// TwinCAT 3 PLC project LineaBosch5PLC
// Title: LineaBosch5
// Company: Normagrup
// ProjectVersion: 1.0
// ProgramVersion: 3.1.4023.0
// libraries:
//   Tc2_Standard, * (Beckhoff Automation GmbH)
//   Tc2_System, * (Beckhoff Automation GmbH)
//   Tc2_Utilities, * (Beckhoff Automation GmbH)
//   Tc3_Module, * (Beckhoff Automation GmbH)
// project tree:
//   DUTs/ ResultadoCiclo.TcDUT
//   GVLs/ GVL.TcGVL
//   / PlcTask.TcTTO
//   POUs/ ControlDescensoFin.TcPOU, ControlElevadorInicio.TcPOU, MAIN.TcPOU, PuestoAutomatico.TcPOU, PuestoTester.TcPOU, PuestoManual.TcPOU, PuestoManualV2.TcPOU, PuestoCupula.TcPOU, Seguridad.TcPOU
// real-time tasks:
//   TASK PlcTask: cycle T#10ms, priority 20, ADS port 350
//   TASK PlcTask1: cycle T#10ms, priority 21, ADS port 351
// I/O:
//   DEVICE Dispositivo 1 (EtherCAT), AmsNetId 5.97.60.79.2.1
//     CabeceraPLC [EK1200-5000 EtherCAT Power supply (2A E-Bus)]
//       Terminal 2 (EL1809) [EL1809 16Ch. Dig. Input 24V, 3ms]
//       Terminal 3 (EL2809) [EL2809 16Ch. Dig. Output 24V, 0.5A]
//       Terminal 4 (EK1110) [EK1110 EtherCAT extension]
//     FinlineaCinta [xFC01 - Rexroth mode]
//     FinLineaVertical [xFC01 - Rexroth mode]
//     CintaLineaSuperior [xFC01 - Rexroth mode]
//     Terminal89 [EK1100 EtherCAT Coupler (2A E-Bus)]
//       Terminal 9 (EL1809) [EL1809 16Ch. Dig. Input 24V, 3ms]
//       Terminal 10 (EL2809) [EL2809 16Ch. Dig. Output 24V, 0.5A]
//       Terminal 31 (EL9011) [EL9011 End Terminal]
//     Valvulas89 [EX260-SEC3 EtherCAT SI Unit (16DO_PNP) Rev1.2]
//     Terminal67 [EK1100 EtherCAT Coupler (2A E-Bus)]
//       Terminal 13 (EL1809) [EL1809 16Ch. Dig. Input 24V, 3ms]
//       Terminal 14 (EL2809) [EL2809 16Ch. Dig. Output 24V, 0.5A]
//       Terminal 32 (EL9011) [EL9011 End Terminal]
//     Valvulas67 [EX260-SEC3 EtherCAT SI Unit (16DO_PNP) Rev1.2]
//     Terminal45 [EK1100 EtherCAT Coupler (2A E-Bus)]
//       Terminal 17 (EL1809) [EL1809 16Ch. Dig. Input 24V, 3ms]
//       Terminal 18 (EL2809) [EL2809 16Ch. Dig. Output 24V, 0.5A]
//       Terminal 33 (EL9011) [EL9011 End Terminal]
//     Valvulas45 [EX260-SEC3 EtherCAT SI Unit (16DO_PNP) Rev1.2]
//     Terminales23 [EK1100 EtherCAT Coupler (2A E-Bus)]
//       Terminal 21 (EL1809) [EL1809 16Ch. Dig. Input 24V, 3ms]
//       Terminal 22 (EL2809) [EL2809 16Ch. Dig. Output 24V, 0.5A]
//       Terminal 34 (EL9011) [EL9011 End Terminal]
//     Valvulas23 [EX260-SEC3 EtherCAT SI Unit (16DO_PNP) Rev1.2]
//     Terminal1 [EK1100 EtherCAT Coupler (2A E-Bus)]
//       Terminal 25 (EL2809) [EL2809 16Ch. Dig. Output 24V, 0.5A]
//       Terminal 26 (EL1809) [EL1809 16Ch. Dig. Input 24V, 3ms]
//       Terminal 35 (EL9011) [EL9011 End Terminal]
//     InicioLineaCinta [xFC01 - Rexroth mode]
//     InicioLineaVertical [xFC01 - Rexroth mode]
//     CintaLineaInferior [xFC01 - Rexroth mode]
//     Valvulas1 [EX260-SEC3 EtherCAT SI Unit (16DO_PNP) Rev1.2]
//   DEVICE Dispositivo 4 (NOV-DP-RAM)
//   DEVICE Dispositivo 6 (RT-Ethernet Protocol), AmsNetId 5.97.60.79.7.1
// variable links:
//   LineaBosch5PLC/LineaBosch5PLC Instance <-> Device 1 (EtherCAT)/CabeceraPLC/Term 2 (EL1809)
//     PlcTask Inputs/GVL.ElevadorFinLinea.PresenciaCintaAbajo <-> Channel 6/Input
//     PlcTask Inputs/GVL.ElevadorFinLinea.PresenciaCintaArriba <-> Channel 7/Input
//     PlcTask Inputs/GVL.ElevadorFinLinea.PulsadorBajar <-> Channel 4/Input
//     PlcTask Inputs/GVL.ElevadorFinLinea.PulsadorSubir <-> Channel 3/Input
//     PlcTask Inputs/GVL.ElevadorFinLinea.SensorAbajo <-> Channel 9/Input
//     PlcTask Inputs/GVL.ElevadorFinLinea.SensorArriba <-> Channel 8/Input
//     PlcTask Inputs/GVL.Elevadorfin1_Presencia <-> Channel 12/Input
//     PlcTask Inputs/GVL.Elevadorfin2_Presencia <-> Channel 14/Input
//     PlcTask Inputs/MAIN.ControlSeguridad.CuadroPrincipalAutomatico <-> Channel 1/Input
//     PlcTask Inputs/MAIN.ControlSeguridad.CuadroPrincipalRunStop <-> Channel 2/Input
//     PlcTask Inputs/MAIN.ControlSeguridad.SeguridadSetas <-> Channel 5/Input
//   LineaBosch5PLC/LineaBosch5PLC Instance <-> Device 1 (EtherCAT)/CabeceraPLC/Term 3 (EL2809)
//     PlcTask Outputs/GVL.SemaforoAmarillo <-> Channel 14/Output
//     PlcTask Outputs/GVL.SemaforoRojo <-> Channel 15/Output
//     PlcTask Outputs/GVL.SemaforoVerde <-> Channel 16/Output
//   LineaBosch5PLC/LineaBosch5PLC Instance <-> Device 1 (EtherCAT)/CintaLineaInferior
//     PlcTask Outputs/MAIN.ControlSeguridad.MotorInferior_Command <-> RxPDO5/Control Word
//     PlcTask Outputs/MAIN.ControlSeguridad.MotorInferior_Freq <-> RxPDO5/Frequency Command
//   LineaBosch5PLC/LineaBosch5PLC Instance <-> Device 1 (EtherCAT)/CintaLineaSuperior
//     PlcTask Outputs/MAIN.ControlSeguridad.MotorSuperior_Command <-> RxPDO5/Control Word
//     PlcTask Outputs/MAIN.ControlSeguridad.MotorSuperior_Freq <-> RxPDO5/Frequency Command
//   LineaBosch5PLC/LineaBosch5PLC Instance <-> Device 1 (EtherCAT)/FinLineaVertical
//     PlcTask Outputs/GVL.ElevadorFinLinea.MotorElevacion_Command <-> RxPDO5/Control Word
//     PlcTask Outputs/GVL.ElevadorFinLinea.MotorElevacion_Freq <-> RxPDO5/Frequency Command
//   LineaBosch5PLC/LineaBosch5PLC Instance <-> Device 1 (EtherCAT)/FinlineaCinta
//     PlcTask Outputs/GVL.ElevadorFinLinea.MotorExtraccion_Command <-> RxPDO5/Control Word
//     PlcTask Outputs/GVL.ElevadorFinLinea.MotorExtraccion_Freq <-> RxPDO5/Frequency Command
//   LineaBosch5PLC/LineaBosch5PLC Instance <-> Device 1 (EtherCAT)/InicioLineaCinta
//     PlcTask Outputs/GVL.ElevadorInicioLinea.MotorExtraccion_Command <-> RxPDO5/Control Word
//     PlcTask Outputs/GVL.ElevadorInicioLinea.MotorExtraccion_Freq <-> RxPDO5/Frequency Command
//   LineaBosch5PLC/LineaBosch5PLC Instance <-> Device 1 (EtherCAT)/InicioLineaVertical
//     PlcTask Outputs/GVL.ElevadorInicioLinea.MotorElevacion_Command <-> RxPDO5/Control Word
//     PlcTask Outputs/GVL.ElevadorInicioLinea.MotorElevacion_Freq <-> RxPDO5/Frequency Command
//   LineaBosch5PLC/LineaBosch5PLC Instance <-> Device 1 (EtherCAT)/Terminal1/Term 26 (EL1809)
//     PlcTask Inputs/GVL.ElevadorInicioLinea.PresenciaCintaAbajo <-> Channel 10/Input
//     PlcTask Inputs/GVL.ElevadorInicioLinea.PresenciaCintaArriba <-> Channel 9/Input
//     PlcTask Inputs/GVL.ElevadorInicioLinea.PulsadorBajar <-> Channel 2/Input
//     PlcTask Inputs/GVL.ElevadorInicioLinea.PulsadorSubir <-> Channel 1/Input
//     PlcTask Inputs/GVL.ElevadorInicioLinea.SensorAbajo <-> Channel 4/Input
//     PlcTask Inputs/GVL.ElevadorInicioLinea.SensorArriba <-> Channel 3/Input
//     PlcTask Inputs/GVL.ElevadorInicioLinea.SensorPaletEnEspera <-> Channel 7/Input
//     PlcTask Inputs/GVL.Elevadorinicio1_Presencia <-> Channel 6/Input
//     PlcTask Inputs/GVL.Elevadorinicio2_Presencia <-> Channel 8/Input
//     PlcTask Inputs/GVL.Puesto11_Presencia <-> Channel 11/Input
//     PlcTask Inputs/GVL.Puesto12_Presencia <-> Channel 13/Input
//   LineaBosch5PLC/LineaBosch5PLC Instance <-> Device 1 (EtherCAT)/Terminal45/Term 17 (EL1809)
//     PlcTask Inputs/GVL.Puesto41_Presencia <-> Channel 3/Input
//     PlcTask Inputs/GVL.Puesto42_Presencia <-> Channel 4/Input
//     PlcTask Inputs/GVL.Puesto51_Presencia <-> Channel 11/Input
//     PlcTask Inputs/GVL.Puesto52_Presencia <-> Channel 12/Input
//   LineaBosch5PLC/LineaBosch5PLC Instance <-> Device 1 (EtherCAT)/Terminal67/Term 13 (EL1809)
//     PlcTask Inputs/GVL.Puesto61_Presencia <-> Channel 3/Input
//     PlcTask Inputs/GVL.Puesto62_Presencia <-> Channel 4/Input
//     PlcTask Inputs/GVL.Puesto71_Presencia <-> Channel 11/Input
//     PlcTask Inputs/GVL.Puesto72_Presencia <-> Channel 12/Input
//     PlcTask Inputs/GVL.Puesto71_Bypass <-> Channel 9/Input
//     PlcTask Inputs/GVL.Puesto71_Pulsador <-> Channel 10/Input
//     PlcTask Inputs/GVL.Puesto72.Fail <-> Channel 13/Input
//     PlcTask Inputs/GVL.Puesto72.Pass <-> Channel 14/Input
//     PlcTask Inputs/GVL.Puesto72.SelectorByPass <-> Channel 15/Input
//     PlcTask Inputs/GVL.Puesto72_PresenciaPieza <-> Channel 16/Input
//   LineaBosch5PLC/LineaBosch5PLC Instance <-> Device 1 (EtherCAT)/Terminal67/Term 14 (EL2809)
//     PlcTask Outputs/GVL.Puesto72.Ready <-> Channel 9/Output
//     PlcTask Outputs/GVL.Puesto72_Actuador <-> Channel 10/Output
//   LineaBosch5PLC/LineaBosch5PLC Instance <-> Device 1 (EtherCAT)/Terminal89/Term 10 (EL2809)
//     PlcTask Outputs/GVL.Puesto81.LuzRoja <-> Channel 1/Output
//   LineaBosch5PLC/LineaBosch5PLC Instance <-> Device 1 (EtherCAT)/Terminal89/Term 9 (EL1809)
//     PlcTask Inputs/GVL.Puesto81_Presencia <-> Channel 3/Input
//     PlcTask Inputs/GVL.Puesto82_Presencia <-> Channel 4/Input
//     PlcTask Inputs/GVL.Puesto91_Presencia <-> Channel 12/Input
//     PlcTask Inputs/GVL.Puesto92_Presencia <-> Channel 11/Input
//     PlcTask Inputs/GVL.Puesto81_Pulsador <-> Channel 5/Input
//   LineaBosch5PLC/LineaBosch5PLC Instance <-> Device 1 (EtherCAT)/Terminales23/Term 21 (EL1809)
//     PlcTask Inputs/GVL.Puesto21_Presencia <-> Channel 3/Input
//     PlcTask Inputs/GVL.Puesto22_Presencia <-> Channel 4/Input
//     PlcTask Inputs/GVL.Puesto31_Presencia <-> Channel 11/Input
//     PlcTask Inputs/GVL.Puesto32_Presencia <-> Channel 12/Input
//   LineaBosch5PLC/LineaBosch5PLC Instance <-> Device 1 (EtherCAT)/Valvulas1
//     PlcTask Outputs/GVL.TerminalValvulas1 <-> Byte 0/Output
//   LineaBosch5PLC/LineaBosch5PLC Instance <-> Device 1 (EtherCAT)/Valvulas23
//     PlcTask Outputs/GVL.TerminalValvulas23 <-> Byte 0/Output
//   LineaBosch5PLC/LineaBosch5PLC Instance <-> Device 1 (EtherCAT)/Valvulas45
//     PlcTask Outputs/GVL.TerminalValvulas45 <-> Byte 0/Output
//   LineaBosch5PLC/LineaBosch5PLC Instance <-> Device 1 (EtherCAT)/Valvulas67
//     PlcTask Outputs/GVL.TerminalValvulas67 <-> Byte 0/Output
//     PlcTask Outputs/GVL.TerminalValvulas67_2 <-> Byte 1/Output
//   LineaBosch5PLC/LineaBosch5PLC Instance <-> Device 1 (EtherCAT)/Valvulas89
//     PlcTask Outputs/GVL.TerminalValvulas89 <-> Byte 0/Output

CONFIGURATION LineaBosch5PLC
    RESOURCE PLC ON TwinCAT3
        TASK PlcTask(INTERVAL := T#10ms, PRIORITY := 21);
        PROGRAM MAIN WITH PlcTask : MAIN;
    END_RESOURCE
END_CONFIGURATION

// ---- DUTs/ResultadoCiclo.TcDUT
{attribute 'pack_mode' := '1'}
TYPE ResultadoCiclo :
STRUCT
	producto  : STRING[25];
	ciclo: INT;
	hora: DT;
	FalloPuesto: ARRAY[1..18] OF BOOL;
	RetrasoPuesto: ARRAY[1..18] OF INT;
END_STRUCT
END_TYPE

// ---- GVLs/GVL.TcGVL
VAR_GLOBAL
	
	
	SeguridadOK :BOOL;
	ModoRun: BOOL;
	ModoAutomatico :BOOL;
	ModoDobleCarga :BOOL := FALSE;
	
	SemaforoRojo AT %Q* :BOOL;
	SemaforoAmarillo AT %Q* :BOOL;
	SemaforoVerde AT %Q* :BOOL;
	
	FinTiempo :BOOL;
	FinCiclo:BOOL;
	
	TiempoDeCiclo: INT := 20;   //segundos de tiempo de ciclo
	VelocidadCinta: UINT := 50; //Velocidad motores cinta en hercios

	FalloPallet: ARRAY[1..18] OF BOOL;

	HoraActual :DT;
	fbLocalTime     : FB_LocalSystemTime;

	
	
	
	TerminalValvulas1 AT %Q*: USINT;
	TerminalValvulas23 AT %Q* : USINT;
	TerminalValvulas45 AT %Q*: USINT;
	TerminalValvulas67 AT %Q* : USINT;
	TerminalValvulas67_2 AT %Q* : USINT;
	TerminalValvulas89 AT %Q* : USINT;
			
	
	Puesto11_Centrador AT %Q* :BOOL;
	Puesto11_stoper AT %Q*:BOOL;
	Puesto12_centrador AT %Q*: BOOL; 
	Puesto12_stoper AT %Q*:BOOL;
	Puesto21_centrador AT %Q*: BOOL; 
	Puesto21_stoper AT %Q*:BOOL;
	Puesto22_centrador AT %Q*: BOOL; 
	Puesto22_stoper AT %Q*:BOOL;
	Puesto31_centrador AT %Q*: BOOL; 
	Puesto31_stoper AT %Q*:BOOL;
	Puesto32_centrador AT %Q*: BOOL; 
	Puesto32_stoper AT %Q*:BOOL;
	Puesto41_centrador AT %Q*: BOOL; 
	Puesto41_stoper AT %Q*:BOOL;
	Puesto42_centrador AT %Q*: BOOL; 
	Puesto42_stoper AT %Q*:BOOL;
	Puesto51_centrador AT %Q*: BOOL; 
	Puesto51_stoper AT %Q*:BOOL;
	Puesto52_centrador AT %Q*: BOOL; 
	Puesto52_stoper AT %Q*:BOOL;
	Puesto61_centrador AT %Q*: BOOL; 
	Puesto61_stoper AT %Q*:BOOL;
	Puesto62_centrador AT %Q*: BOOL; 
	Puesto62_stoper AT %Q*:BOOL;
	Puesto71_centrador AT %Q*: BOOL; 
	Puesto71_stoper AT %Q*:BOOL;
	Puesto72_centrador AT %Q*: BOOL; 
	Puesto72_stoper AT %Q*:BOOL;
	Puesto81_centrador AT %Q*: BOOL; 
	Puesto81_stoper AT %Q*:BOOL;
	Puesto82_centrador AT %Q*: BOOL; 
	Puesto82_stoper AT %Q*:BOOL;
	Puesto91_centrador AT %Q*: BOOL; 
	Puesto91_stoper AT %Q*:BOOL;
	Puesto92_centrador AT %Q*: BOOL; 
	Puesto92_stoper AT %Q*:BOOL;
	
	Puesto71_Actuador AT %Q* :BOOL;
	Puesto72_Actuador AT %Q* :BOOL;
	Puesto72_LuzVerde AT %Q* :BOOL;
	

	
	Puesto11_Presencia AT %I* :BOOL;
	Puesto12_Presencia AT %I* :BOOL;
	Puesto21_Presencia AT %I* :BOOL;
	Puesto22_Presencia AT %I* :BOOL;
	Puesto31_Presencia AT %I* :BOOL;
	Puesto32_Presencia AT %I* :BOOL;
	Puesto41_Presencia AT %I* :BOOL;
	Puesto42_Presencia AT %I* :BOOL;
	Puesto51_Presencia AT %I* :BOOL;
	Puesto52_Presencia AT %I* :BOOL;
	Puesto61_Presencia AT %I* :BOOL;
	Puesto62_Presencia AT %I* :BOOL;
	Puesto71_Presencia AT %I* :BOOL;
	Puesto72_Presencia AT %I* :BOOL;
	Puesto81_Presencia AT %I* :BOOL;
	Puesto82_Presencia AT %I* :BOOL;
	Puesto91_Presencia AT %I* :BOOL;
	Puesto92_Presencia AT %I* :BOOL;
	
	Puesto61_Bypass AT %I* :BOOL;
	Puesto71_Pulsador AT %I* :BOOL;
	Puesto71_Bypass AT %I* :BOOL;
	Puesto72_PresenciaPieza AT %I* :BOOL;
	Puesto81_Pulsador AT %I* :BOOL;

	Elevadorinicio1_Presencia AT %I* :BOOL;
	Elevadorinicio2_Presencia AT %I* :BOOL;
	Elevadorfin1_Presencia AT %I* :BOOL;
	Elevadorfin2_Presencia AT %I* :BOOL;

	
	Puesto11: PuestoManual;
    Puesto12: PuestoManual;
    Puesto21: PuestoManual;
    Puesto22: PuestoManual;
    Puesto31: PuestoManual;
	Puesto32: PuestoManual;
    Puesto41: PuestoManual;
	Puesto42: PuestoManual;
    Puesto51: PuestoManual;
	Puesto52: PuestoManual;
    Puesto61: PuestoManual;
	Puesto62: PuestoManual;
    Puesto71: PuestoCupula;
	Puesto72: PuestoAutomatico;
    Puesto81: PuestoManual;
	Puesto82: PuestoManual;
    Puesto91: PuestoManual;
	Puesto92: PuestoManualV2;
	

	

	ElevadorFinLinea: ControlDescensoFin;
	ElevadorInicioLinea: ControlElevadorInicio;
	
END_VAR

VAR_GLOBAL PERSISTENT
	Producto : STRING[30] := 'SINDEFINIR';
	Est_Resultados : ARRAY[1..3000] OF ResultadoCiclo;
	PunteroEst: INT := 1;
END_VAR

// ---- POUs/MAIN.TcPOU
PROGRAM MAIN
VAR
	ControlSeguridad: Seguridad;
	ElevadorFinLleno : BOOL;
	ElevadorInicioLleno :BOOL;
	ElevadorInicioPuedeExtraer :BOOL;
	FalloTest :BOOL;

	fbTime   : FB_LocalSystemTime := ( bEnable := TRUE, dwCycle := 100 );
	
	Semaforo: USINT;
	EstadoPuestos: DINT;
	
END_VAR

	
ControlSeguridad();
fbTime();
gvl.HoraActual := SYSTEMTIME_TO_DT(fbTime.systemTime);

///PUESTO 1 -----------------------------------

Puesto12 ( Enable:= gvl.ModoRun, Reset := FALSE,SensorPallet:= gvl.Puesto12_Presencia, 
		Centrador => gvl.Puesto12_centrador, StopperOFF => gvl.Puesto12_stoper,
FinCiclo := gvl.FinCiclo, NumeroDePuesto :=1   );


///PUESTO 2 -----------------------------------
Puesto21 ( Enable:= gvl.ModoRun, Reset := FALSE,SensorPallet:= gvl.Puesto21_Presencia, 
		Centrador => gvl.Puesto21_centrador, StopperOFF => gvl.Puesto21_stoper,
FinCiclo := gvl.FinCiclo, NumeroDePuesto :=2   );
Puesto22 ( Enable:= gvl.ModoRun, Reset := FALSE,SensorPallet:= gvl.Puesto22_Presencia, 
		Centrador => gvl.Puesto22_centrador, StopperOFF => gvl.Puesto22_stoper,
FinCiclo := gvl.FinCiclo, NumeroDePuesto :=3   );

///PUESTO 3 -----------------------------------
Puesto31 ( Enable:= gvl.ModoRun, Reset := FALSE,SensorPallet:= gvl.Puesto31_Presencia, 
		Centrador => gvl.Puesto31_centrador, StopperOFF => gvl.Puesto31_stoper,
FinCiclo := gvl.FinCiclo, NumeroDePuesto :=4   );
Puesto32 ( Enable:= gvl.ModoRun, Reset := FALSE,SensorPallet:= gvl.Puesto32_Presencia, 
		Centrador => gvl.Puesto32_centrador, StopperOFF => gvl.Puesto32_stoper,
FinCiclo := gvl.FinCiclo, NumeroDePuesto :=5   );

///PUESTO 4 -----------------------------------
Puesto41 ( Enable:= gvl.ModoRun, Reset := FALSE,SensorPallet:= gvl.Puesto41_Presencia, 
		Centrador => gvl.Puesto41_centrador, StopperOFF => gvl.Puesto41_stoper,
FinCiclo := gvl.FinCiclo, NumeroDePuesto :=6   );
Puesto42 ( Enable:= gvl.ModoRun, Reset := FALSE,SensorPallet:= gvl.Puesto42_Presencia, 
		Centrador => gvl.Puesto42_centrador, StopperOFF => gvl.Puesto42_stoper,
FinCiclo := gvl.FinCiclo, NumeroDePuesto :=7   );

///PUESTO 5 -----------------------------------
Puesto51 ( Enable:= gvl.ModoRun, Reset := FALSE,SensorPallet:= gvl.Puesto51_Presencia, 
		Centrador => gvl.Puesto51_centrador, StopperOFF => gvl.Puesto51_stoper,
FinCiclo := gvl.FinCiclo, NumeroDePuesto :=8   );
Puesto52 ( Enable:= gvl.ModoRun, Reset := FALSE,SensorPallet:= gvl.Puesto52_Presencia, 
		Centrador => gvl.Puesto52_centrador, StopperOFF => gvl.Puesto52_stoper,
FinCiclo := gvl.FinCiclo, NumeroDePuesto :=9   );

///PUESTO 6 -----------------------------------
Puesto61 ( Enable:= gvl.ModoRun, Reset := FALSE,SensorPallet:= gvl.Puesto61_Presencia, 
		Centrador => gvl.Puesto61_centrador, StopperOFF => gvl.Puesto61_stoper,
FinCiclo := gvl.FinCiclo, NumeroDePuesto :=10   );
Puesto62 ( Enable:= gvl.ModoRun, Reset := FALSE,SensorPallet:= gvl.Puesto62_Presencia, 
		Centrador => gvl.Puesto62_centrador, StopperOFF => gvl.Puesto62_stoper,
FinCiclo := gvl.FinCiclo, NumeroDePuesto :=11   );

///PUESTO 7 -----------------------------------
//Puesto71 ( Enable:= gvl.ModoRun, Reset := FALSE,SensorPallet:= gvl.Puesto71_Presencia, 
//		Centrador => gvl.Puesto71_centrador, StopperOFF => gvl.Puesto71_stoper,
//FinCiclo := gvl.FinCiclo, NumeroDePuesto :=12   );

///*****************************************************

Puesto71 ( Enable:= gvl.ModoRun, Reset :=FALSE,SensorPallet:= gvl.Puesto71_Presencia, 
			sensorpieza1 :=TRUE, SelectorByPass := gvl.Puesto71_Bypass,
		Centrador => gvl.Puesto71_centrador, StopperOFF => gvl.Puesto71_stoper,
		FinCiclo := gvl.FinCiclo , NumeroDePuesto :=12  );
gvl.Puesto71_Actuador:= Puesto71.Actuador;

//***********************************************************



//Puesto del Test 
Puesto72 ( Enable:= gvl.ModoRun, Reset :=FALSE,SensorPallet:= gvl.Puesto72_Presencia, 
			sensorpieza1 := gvl.Puesto72_presenciapieza, Centrador => gvl.Puesto72_centrador, StopperOFF => gvl.Puesto72_stoper,
		FinCiclo := gvl.FinCiclo , NumeroDePuesto :=13  );
gvl.Puesto72_Actuador := gvl.Puesto72.Ready; ///gvl.Puesto72_centrador AND gvl.Puesto72_PresenciaPieza ;
gvl.Puesto72_LuzVerde := Puesto72.Ready;


///PUESTO 8 -----------------------------------
Puesto81 ( Enable:= gvl.ModoRun, Reset := FALSE,SensorPallet:= gvl.Puesto81_Presencia, 
		Centrador => gvl.Puesto81_centrador, StopperOFF => gvl.Puesto81_stoper,
		pulsador1:= gvl.Puesto81_Pulsador,
FinCiclo := gvl.FinCiclo, NumeroDePuesto :=14   );

Puesto82 ( Enable:= gvl.ModoRun, Reset := FALSE,SensorPallet:= gvl.Puesto82_Presencia, 
		Centrador => gvl.Puesto82_centrador, StopperOFF => gvl.Puesto82_stoper,
FinCiclo := gvl.FinCiclo, NumeroDePuesto :=15  );


///PUESTO 9 -----------------------------------
Puesto91 ( Enable:= gvl.ModoRun, Reset := FALSE,SensorPallet:= gvl.Puesto91_Presencia, 
		Centrador => gvl.Puesto91_centrador, StopperOFF => gvl.Puesto91_stoper,
FinCiclo := gvl.FinCiclo, NumeroDePuesto :=16   );



/// ojo modo doble carga 
gvl.ModoDobleCarga := TRUE;

Puesto11 ( Enable:= gvl.ModoRun, Reset := FALSE,SensorPallet:= gvl.Puesto11_Presencia, 
		Centrador => gvl.Puesto11_centrador, StopperOFF => gvl.Puesto11_stoper,
FinCiclo := gvl.FinCiclo, NumeroDePuesto :=17  );


Puesto92 ( Enable:= gvl.ModoRun, Reset := FALSE,SensorPallet:= gvl.Puesto92_Presencia, 
		Centrador => gvl.Puesto92_centrador, StopperOFF => gvl.Puesto92_stoper,
FinCiclo := gvl.FinCiclo, NumeroDePuesto :=18 , ModoDoble := gvl.ModoDobleCarga  );


/// CONTROL ELEVADORES

IF gvl.ModoDobleCarga = TRUE THEN
	ElevadorFinLleno := gvl.Elevadorfin1_Presencia AND gvl.Elevadorfin2_Presencia;
	ElevadorInicioLleno := gvl.Elevadorinicio1_Presencia AND gvl.Elevadorinicio2_Presencia;
	ElevadorInicioPuedeExtraer := Puesto11.EsperandoPalet AND Puesto12.EsperandoPalet;
ELSE
	ElevadorFinLleno := gvl.Elevadorfin1_Presencia;
	ElevadorInicioLleno := gvl.Elevadorinicio1_Presencia;
	ElevadorInicioPuedeExtraer := Puesto11.EsperandoPalet;
END_IF

ElevadorInicioLinea( Enabled:= gvl.ModoRun, SeguridadOK:= GVL.SeguridadOK,
					SensorPaletFuera := Puesto11.SensorPallet,
					SensorPaletDentro := ElevadorInicioLleno,
					 PuedeExtraer := Puesto11.EsperandoPalet AND NOT Puesto12.EsperandoPalet);
					 
ElevadorFinLinea( Enabled:= gvl.ModoRun, SeguridadOK:= GVL.SeguridadOK, 
				SensorPaletDentro := ElevadorFinLleno,
				SensorPaletFuera := gvl.Elevadorfin2_Presencia,
				PuedeExtraer := TRUE);

TerminalValvulas1.0 := ElevadorInicioLinea.StopperOFF;
TerminalValvulas1.1 := gvl.Puesto11_stoper;
TerminalValvulas1.2 := gvl.Puesto12_stoper;
TerminalValvulas1.3 := gvl.Puesto11_centrador;
TerminalValvulas1.4 := gvl.Puesto12_centrador;

TerminalValvulas23.0 := gvl.Puesto21_stoper;
TerminalValvulas23.1 := gvl.Puesto22_stoper;
TerminalValvulas23.2 := gvl.Puesto31_stoper;
TerminalValvulas23.3 := gvl.Puesto32_stoper;
TerminalValvulas23.4 := gvl.Puesto21_centrador;
TerminalValvulas23.5 := gvl.Puesto22_centrador;
TerminalValvulas23.6 := gvl.Puesto31_centrador;
TerminalValvulas23.7 := gvl.Puesto32_centrador;

TerminalValvulas45.0 := gvl.Puesto41_stoper;
TerminalValvulas45.1 := gvl.Puesto42_stoper;
TerminalValvulas45.2 := gvl.Puesto51_stoper;
TerminalValvulas45.3 := gvl.Puesto52_stoper;
TerminalValvulas45.4 := gvl.Puesto41_centrador;
TerminalValvulas45.5 := gvl.Puesto42_centrador;
TerminalValvulas45.6 := gvl.Puesto51_centrador;
TerminalValvulas45.7 := gvl.Puesto52_centrador;

TerminalValvulas67.0 := gvl.Puesto61_stoper;
TerminalValvulas67.1 := gvl.Puesto62_stoper;
TerminalValvulas67.2 := gvl.Puesto71_stoper;
TerminalValvulas67.3 := gvl.Puesto72_stoper;
TerminalValvulas67.4 := gvl.Puesto61_centrador;
TerminalValvulas67.5 := gvl.Puesto62_centrador;
TerminalValvulas67.6 := gvl.Puesto71_centrador;
TerminalValvulas67.7 := gvl.Puesto72_centrador;
TerminalValvulas67_2.0 := gvl.Puesto72_actuador;
TerminalValvulas67_2.1 := gvl.Puesto71_actuador;


TerminalValvulas89.0 := gvl.Puesto81_stoper;
TerminalValvulas89.1 := gvl.Puesto82_stoper;
TerminalValvulas89.2 := gvl.Puesto91_stoper;
TerminalValvulas89.3 := gvl.Puesto92_stoper;
TerminalValvulas89.4 := gvl.Puesto81_centrador;
TerminalValvulas89.5 := gvl.Puesto82_centrador;
TerminalValvulas89.6 := gvl.Puesto91_centrador;
TerminalValvulas89.7 := gvl.Puesto92_centrador;

/// Variables para el HMI
Semaforo.0 := gvl.SemaforoRojo;
Semaforo.1 := gvl.SemaforoAmarillo;
Semaforo.2 := gvl.SemaforoVerde;

 EstadoPuestos.0 := GVL.ElevadorInicioLinea.Ready;
 EstadoPuestos.1 := GVL.Puesto11.FinPuesto;
 EstadoPuestos.2 := GVL.Puesto12.FinPuesto;
 EstadoPuestos.3 := GVL.Puesto21.FinPuesto;
 EstadoPuestos.4 := GVL.Puesto22.FinPuesto ;
 EstadoPuestos.5 := GVL.Puesto31.FinPuesto;
 EstadoPuestos.6 := GVL.Puesto32.FinPuesto;
 EstadoPuestos.7 := GVL.Puesto41.FinPuesto;
 EstadoPuestos.8 := GVL.Puesto42.FinPuesto ;
 EstadoPuestos.9 := GVL.Puesto51.FinPuesto ;
 EstadoPuestos.10 := GVL.Puesto52.FinPuesto ;
 EstadoPuestos.11 := GVL.Puesto61.FinPuesto ;
 EstadoPuestos.12 := GVL.Puesto62.FinPuesto ;
 EstadoPuestos.13 := GVL.Puesto71.FinPuesto ;
 EstadoPuestos.14 := GVL.Puesto72.FinPuesto ;
 EstadoPuestos.15 := GVL.Puesto81.FinPuesto ;
 EstadoPuestos.16 := GVL.Puesto82.FinPuesto ;
 EstadoPuestos.17 := GVL.Puesto91.FinPuesto ;
 EstadoPuestos.18 := GVL.Puesto92.FinPuesto ;
 EstadoPuestos.19 := GVL.ElevadorFinLinea.Ready;

END_PROGRAM

// ---- POUs/Seguridad.TcPOU
FUNCTION_BLOCK Seguridad
VAR_INPUT
	
	CuadroPrincipalRunStop AT%I*:BOOL;
	CuadroPrincipalAutomatico AT%I*:BOOL;
	SeguridadSetas AT%I*:BOOL;
END_VAR
VAR_OUTPUT
	CuadroLedVerde AT%Q*:BOOL;
	CuadroLedAmarillo AT%Q*:BOOL;
	
	MotorSuperior_Freq  AT%Q*: UINT;
	MotorSuperior_Command AT%Q*: INT;
		
	MotorInferior_Freq  AT%Q*: UINT;
	MotorInferior_Command AT%Q*: INT;
	
	LineaReady :BOOL;
	FinTiempoTON :TON;
	
	
	
END_VAR
VAR
	FlancoRunStop:R_TRIG;
	TempCiclo:TON;
	TempRetraso:TON;
	Resultados : ResultadoCiclo;

	puesto: INT;
	Falso: BOOL;
END_VAR

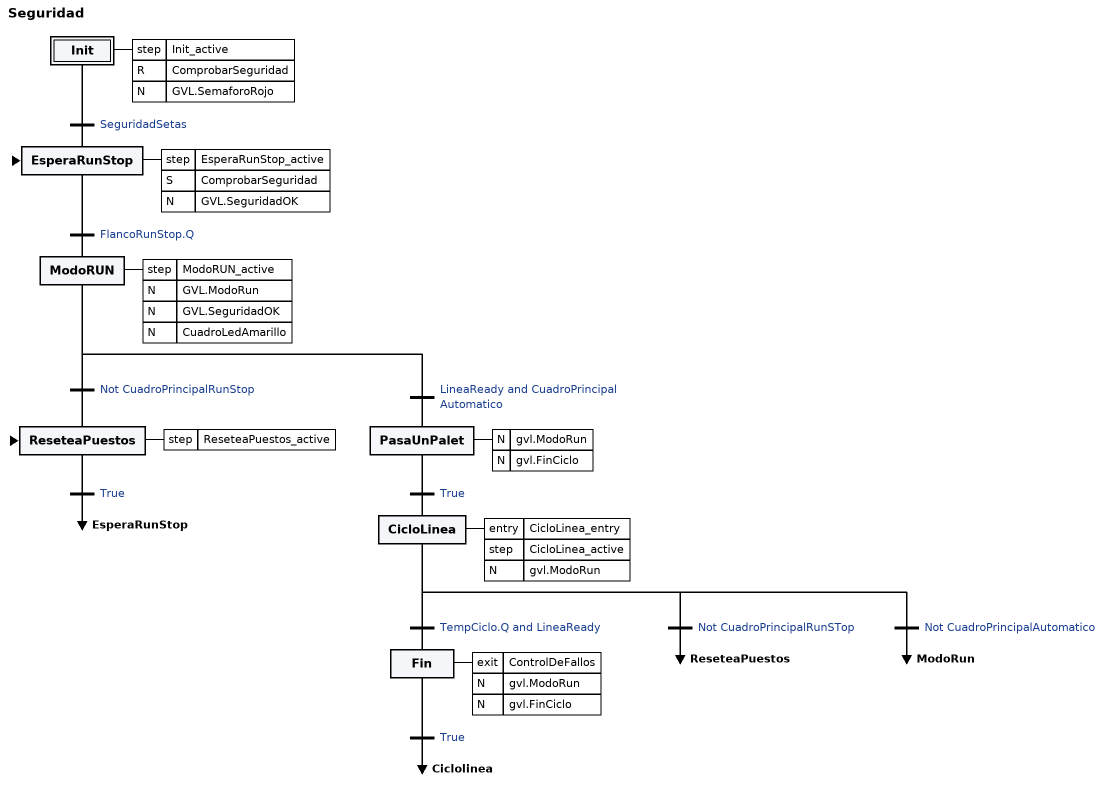
INITIAL_STEP Init:
    Init_active(N);  // step action
    ComprobarSeguridad(R);
    GVL.SemaforoRojo(N);
END_STEP
TRANSITION FROM Init TO EsperaRunStop
    := SeguridadSetas;
END_TRANSITION
STEP EsperaRunStop:  // min time T#1s
    EsperaRunStop_active(N);  // step action
    ComprobarSeguridad(S);
    GVL.SeguridadOK(N);
END_STEP
TRANSITION FROM EsperaRunStop TO ModoRUN
    := FlancoRunStop.Q;
END_TRANSITION
STEP ModoRUN:  // min time T#1s
    ModoRUN_active(N);  // step action
    GVL.ModoRun(N);
    GVL.SeguridadOK(N);
    CuadroLedAmarillo(N);
END_STEP
TRANSITION FROM ModoRUN TO ReseteaPuestos
    := Not CuadroPrincipalRunStop;
END_TRANSITION
STEP ReseteaPuestos:  // min time T#1s
    ReseteaPuestos_active(N);  // step action
END_STEP
TRANSITION FROM ReseteaPuestos TO EsperaRunStop
    := True;
END_TRANSITION
TRANSITION FROM ModoRUN TO PasaUnPalet
    := LineaReady and CuadroPrincipalAutomatico;
END_TRANSITION
STEP PasaUnPalet:  // min time T#3s
    gvl.ModoRun(N);
    gvl.FinCiclo(N);
END_STEP
TRANSITION FROM PasaUnPalet TO CicloLinea
    := True;
END_TRANSITION
STEP CicloLinea:  // min time T#4s
    CicloLinea_entry(P1);  // entry action
    CicloLinea_active(N);  // step action
    gvl.ModoRun(N);
END_STEP
TRANSITION FROM CicloLinea TO Fin
    := TempCiclo.Q and LineaReady;
END_TRANSITION
STEP Fin:  // min time T#3s
    ControlDeFallos(P0);  // exit action
    gvl.ModoRun(N);
    gvl.FinCiclo(N);
END_STEP
TRANSITION FROM Fin TO Ciclolinea
    := True;
END_TRANSITION
TRANSITION FROM CicloLinea TO ReseteaPuestos
    := Not CuadroPrincipalRunSTop;
END_TRANSITION
TRANSITION FROM CicloLinea TO ModoRun
    := Not CuadroPrincipalAutomatico;
END_TRANSITION

ACTION CicloLinea_active:
TempCiclo(IN:=TRUE);
TempRetraso(IN:=TempCiclo.Q);

gvl.SemaforoVerde := TRUE;

IF (    (ElevadorInicioLinea.Ready OR gvl.ModoDobleCarga)///no esperamos por elevador inicio en modo doble carga
	AND (ElevadorFinLinea.ready OR GVL.Puesto92.EsperandoPalet ) //si el ultimo  puesto no tieen palet no esperamos por elevador fin
	AND GVL.Puesto11.FinPuesto AND
		GVL.Puesto12.FinPuesto AND
		GVL.Puesto21.FinPuesto AND
		GVL.Puesto22.FinPuesto AND
		GVL.Puesto31.FinPuesto AND
		GVL.Puesto32.FinPuesto AND
		GVL.Puesto41.FinPuesto AND
		GVL.Puesto42.FinPuesto AND
		GVL.Puesto51.FinPuesto AND
		GVL.Puesto52.FinPuesto AND
		GVL.Puesto61.FinPuesto AND
		GVL.Puesto62.FinPuesto AND
		GVL.Puesto71.FinPuesto AND
		GVL.Puesto72.FinPuesto AND
		GVL.Puesto81.FinPuesto AND
		GVL.Puesto82.FinPuesto AND
		GVL.Puesto91.FinPuesto AND
		(gvl.Puesto81.LuzRoja = FALSE) AND
		(GVL.Puesto92.FinPuesto OR gvl.ModoDobleCarga))
THEN
		LineaReady := TRUE;
		gvl.SemaforoAmarillo :=  FALSE;
ELSE 
	    LineaReady := FALSE;
		gvl.SemaforoAmarillo := TempCiclo.Q;
END_IF


IF TempCiclo.Q AND NOT Lineaready THEN

		IF NOT  GVL.Puesto11.FinPuesto THEN gvl.Est_Resultados[gvl.PunteroEst].RetrasoPuesto[1] := TIME_TO_INT(TempRetraso.ET)/1000; END_IF 
		IF NOT 	GVL.Puesto12.FinPuesto THEN gvl.Est_Resultados[gvl.PunteroEst].RetrasoPuesto[2] := TIME_TO_INT(TempRetraso.ET); END_IF 
		if not 	GVL.Puesto21.FinPuesto then gvl.Est_Resultados[gvl.PunteroEst].RetrasoPuesto[3] := TIME_TO_INT(TempRetraso.ET); END_IF 
		if not 	GVL.Puesto22.FinPuesto then gvl.Est_Resultados[gvl.PunteroEst].RetrasoPuesto[4] := TIME_TO_INT(TempRetraso.ET); END_IF 
		if not 	GVL.Puesto31.FinPuesto then gvl.Est_Resultados[gvl.PunteroEst].RetrasoPuesto[5] := TIME_TO_INT(TempRetraso.ET); END_IF 
		if not 	GVL.Puesto32.FinPuesto then gvl.Est_Resultados[gvl.PunteroEst].RetrasoPuesto[6] := TIME_TO_INT(TempRetraso.ET); END_IF 
		if not 	GVL.Puesto41.FinPuesto then gvl.Est_Resultados[gvl.PunteroEst].RetrasoPuesto[7] := TIME_TO_INT(TempRetraso.ET); END_IF 
		if not 	GVL.Puesto42.FinPuesto then gvl.Est_Resultados[gvl.PunteroEst].RetrasoPuesto[8] := TIME_TO_INT(TempRetraso.ET); END_IF 
		if not 	GVL.Puesto51.FinPuesto then gvl.Est_Resultados[gvl.PunteroEst].RetrasoPuesto[9] := TIME_TO_INT(TempRetraso.ET); END_IF 
		if not 	GVL.Puesto52.FinPuesto then gvl.Est_Resultados[gvl.PunteroEst].RetrasoPuesto[10] := TIME_TO_INT(TempRetraso.ET); END_IF 
		if not 	GVL.Puesto61.FinPuesto then gvl.Est_Resultados[gvl.PunteroEst].RetrasoPuesto[11] := TIME_TO_INT(TempRetraso.ET); END_IF 
		if not 	GVL.Puesto62.FinPuesto then gvl.Est_Resultados[gvl.PunteroEst].RetrasoPuesto[12] := TIME_TO_INT(TempRetraso.ET); END_IF 
		if not 	GVL.Puesto71.FinPuesto then gvl.Est_Resultados[gvl.PunteroEst].RetrasoPuesto[13] := TIME_TO_INT(TempRetraso.ET); END_IF 
		if not 	GVL.Puesto72.FinPuesto then gvl.Est_Resultados[gvl.PunteroEst].RetrasoPuesto[14] := TIME_TO_INT(TempRetraso.ET); END_IF 
		if not 	GVL.Puesto81.FinPuesto then gvl.Est_Resultados[gvl.PunteroEst].RetrasoPuesto[15] := TIME_TO_INT(TempRetraso.ET); END_IF 
		if not 	GVL.Puesto82.FinPuesto then gvl.Est_Resultados[gvl.PunteroEst].RetrasoPuesto[16] := TIME_TO_INT(TempRetraso.ET); END_IF 
		if not 	GVL.Puesto91.FinPuesto then gvl.Est_Resultados[gvl.PunteroEst].RetrasoPuesto[17] := TIME_TO_INT(TempRetraso.ET); END_IF 
		if not 	GVL.Puesto92.FinPuesto then gvl.Est_Resultados[gvl.PunteroEst].RetrasoPuesto[18] := TIME_TO_INT(TempRetraso.ET); END_IF 

END_IF
END_ACTION

ACTION CicloLinea_entry:
TempCiclo(IN:=FALSE, PT:= DWORD_TO_TIME(  (INT_TO_DWORD(gvl.TiempoDeCiclo) -3)* 1000));
TempRetraso(IN:=FALSE, PT:= T#15M);



gvl.PunteroEst := gvl.PunteroEst +1;
IF gvl.PunteroEst > 1999 THEN
	gvl.PunteroEst := 1;
END_IF


//Creamos un nuevo registros
gvl.Est_Resultados[gvl.PunteroEst].Ciclo := gvl.TiempoDeCiclo;
gvl.Est_Resultados[gvl.PunteroEst].Producto := gvl.Producto;
gvl.Est_Resultados[gvl.PunteroEst].hora := gvl.HoraActual;



FOR puesto := 1 TO 18 DO
	gvl.Est_Resultados[gvl.PunteroEst].FalloPuesto[puesto] := FALSE;
	gvl.Est_Resultados[gvl.PunteroEst].RetrasoPuesto[puesto] := 0;
	
END_FOR
END_ACTION

ACTION ComprobarSeguridad:
IF NOT SeguridadSetas THEN
	SFCReset:=TRUE;
END_IF
END_ACTION

ACTION ControlDeFallos:




//avanzamos el fallo en el palet y guardamos estadistica
FOR puesto := 18 TO 2 BY -1 DO
	gvl.Est_Resultados[gvl.PunteroEst].FalloPuesto[puesto] := gvl.FalloPallet[puesto];
	gvl.FalloPallet[puesto] := gvl.FalloPallet[puesto -1 ];
END_FOR

gvl.FalloPallet[1] := Falso;
END_ACTION

ACTION EsperaRunStop_active:
FlancoRunStop(CLK:=CuadroPrincipalRunStop);

Gvl.SemaforoAmarillo := TRUE;
MotorCintaSuperior(0);
MotorCintaInferior(0);
END_ACTION

ACTION Init_active:
MotorCintaSuperior(0);
MotorCintaInferior(0);
SFCreset := FALSE;
gvl.SemaforoAmarillo :=FALSE;
gvl.SemaforoVerde := FALSE;
END_ACTION

ACTION ModoRUN_active:

TempCiclo(IN:=FALSE);

IF ElevadorFinLinea.Ready THEN
 MotorCintaSuperior(1);
END_IF

gvl.SemaforoAmarillo :=TRUE;

IF ElevadorInicioLinea.EsperandoPalet OR ElevadorInicioLinea.Ready THEN
	MotorCintaInferior(1);
END_IF

IF (ElevadorInicioLinea.Ready AND
	ElevadorFinLinea.ready AND 
	GVL.Puesto12.FinPuesto AND
	GVL.Puesto21.FinPuesto AND
	GVL.Puesto22.FinPuesto AND
	GVL.Puesto31.FinPuesto AND
	GVL.Puesto32.FinPuesto AND
	GVL.Puesto41.FinPuesto AND
	GVL.Puesto42.FinPuesto AND
	GVL.Puesto51.FinPuesto AND
	GVL.Puesto52.FinPuesto AND
	GVL.Puesto61.FinPuesto AND
	GVL.Puesto62.FinPuesto AND
	GVL.Puesto71.FinPuesto AND
	GVL.Puesto72.FinPuesto AND
	GVL.Puesto81.FinPuesto AND
	GVL.Puesto82.FinPuesto AND
	GVL.Puesto91.FinPuesto )
THEN		
		gvl.SemaforoVerde := TRUE;
		LineaReady := TRUE;
			
ELSE
			LineaReady:=FALSE;
			gvl.FinTiempo :=FALSE;
			gvl.SemaforoVerde := FALSE;
END_IF
END_ACTION

METHOD PRIVATE MotorCintaInferior : BOOL
VAR_INPUT
	Direccion: INT;
END_VAR
MotorInferior_Freq := gvl.VelocidadCinta * 100;


MotorInferior_Command := 0;
MotorInferior_Command.7 := 1 ; //Control Word Active


IF Direccion  = 0 THEN
	MotorInferior_Command.3 := 1 ; // Stop according to parameter setting	

ELSIF gvl.ElevadorInicioLinea.PresenciaCintaAbajo AND NOT gvl.ElevadorInicioLinea.SensorAbajo THEN
	// presencia en la salida y el elevador no esta abajo: paramos y ERROR
	MotorInferior_Command.3 := 1 ;
	
ELSIF Direccion  = 1 THEN		
		MotorInferior_Command.2 := 1 ; //1 reversed 0 fordward
		MotorInferior_Command.0 := 1 ; // Run Command active
ELSE
	MotorInferior_Command.3 := 1 ; // Stop according to parameter setting	
END_IF
END_METHOD

METHOD PRIVATE MotorCintaSuperior : BOOL
VAR_INPUT
	Direccion: INT;
END_VAR
MotorSuperior_Freq := gvl.VelocidadCinta * 100;


MotorSuperior_Command := 0;
MotorSuperior_Command.7 := 1 ; //Control Word Active

IF Direccion = 0 THEN
	MotorSuperior_Command.3 := 1 ; // Stop according to parameter setting	
ELSIF gvl.Elevadorfinlinea.PresenciaCintaArriba AND NOT gvl.Elevadorfinlinea.sensorarriba THEN
	//ERROR : palet en la salida y elevador no arriba
	MotorSuperior_Command.3 := 1 ;
ELSIF Direccion  = 1 THEN		
		MotorSuperior_Command.2 := 0 ; //1 reversed 0 fordward
		MotorSuperior_Command.0 := 1 ; // Run Command active
ELSE
	MotorSuperior_Command.3 := 1 ; // Stop according to parameter setting	
END_IF
END_METHOD

ACTION ReseteaPuestos_active:

//Resetea los puestos para pasar un palet


GVL.Puesto11.SFCreset := TRUE;
GVL.Puesto12.SFCreset := TRUE;
GVL.Puesto21.SFCreset := TRUE;
GVL.Puesto22.SFCreset := TRUE;
GVL.Puesto31.sfcreset := TRUE;
GVL.Puesto32.sfcreset := TRUE;
GVL.Puesto41.sfcreset := TRUE;
GVL.Puesto42.sfcreset := TRUE;
GVL.Puesto51.sfcreset := TRUE;
GVL.Puesto52.sfcreset := TRUE;
GVL.Puesto61.sfcreset := TRUE;
GVL.Puesto62.sfcreset := TRUE;
GVL.Puesto71.sfcreset := TRUE;
GVL.Puesto72.sfcreset := TRUE;
GVL.Puesto81.sfcreset := TRUE;
GVL.Puesto82.sfcreset := TRUE;
GVL.Puesto91.sfcreset := TRUE;
GVL.Puesto92.sfcreset := TRUE;

ElevadorInicioLinea.SFCreset := TRUE;
ElevadorFinLinea.SFCreset := TRUE;
END_ACTION

END_FUNCTION_BLOCK

// ---- POUs/PuestoManual.TcPOU
FUNCTION_BLOCK PuestoManual
VAR_INPUT
	SFCreset:BOOL;
	Reset:BOOL;
	Enable:BOOL;
	FinCiclo:BOOL;
	SensorPallet:BOOL;
	Pulsador1 AT %I*:BOOL;
	NumeroDePuesto :INT;
	
END_VAR
VAR_OUTPUT
	StopperOFF AT %Q*:BOOL;
	Centrador AT%Q*:BOOL;
	LuzRoja AT%Q*:BOOL;
	FinPuesto:BOOL;
	SalidaAlarma:BOOL;
	EnMovimiento:BOOL;
	EsperandoPalet :BOOL;
	RetrasoPuesto :INT;
END_VAR
VAR
END_VAR

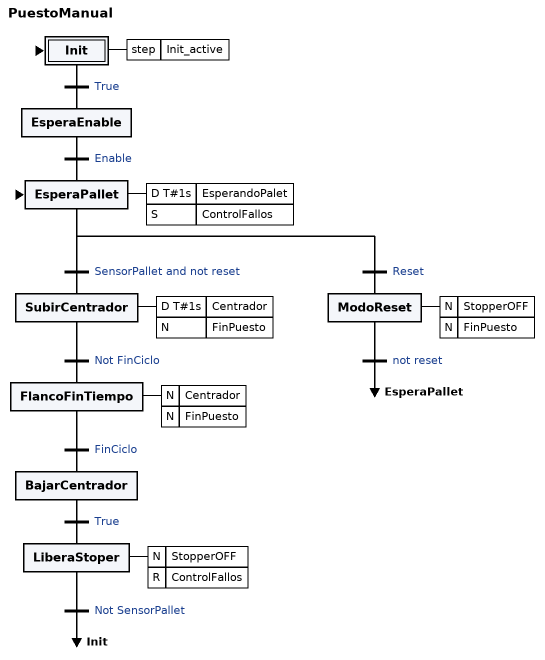
INITIAL_STEP Init:
    Init_active(N);  // step action
END_STEP
TRANSITION FROM Init TO EsperaEnable
    := True;
END_TRANSITION
STEP EsperaEnable:
END_STEP
TRANSITION FROM EsperaEnable TO EsperaPallet
    := Enable;
END_TRANSITION
STEP EsperaPallet:
    EsperandoPalet(D, T#1s);
    ControlFallos(S);
END_STEP
TRANSITION FROM EsperaPallet TO SubirCentrador
    := SensorPallet and not reset;
END_TRANSITION
STEP SubirCentrador:  // min time T#1s
    Centrador(D, T#1s);
    FinPuesto(N);
END_STEP
TRANSITION FROM SubirCentrador TO FlancoFinTiempo
    := Not FinCiclo;
END_TRANSITION
STEP FlancoFinTiempo:
    Centrador(N);
    FinPuesto(N);
END_STEP
TRANSITION FROM FlancoFinTiempo TO BajarCentrador
    := FinCiclo;
END_TRANSITION
STEP BajarCentrador:  // min time T#1s
END_STEP
TRANSITION FROM BajarCentrador TO LiberaStoper
    := True;
END_TRANSITION
TRANSITION FROM EsperaPallet TO ModoReset
    := Reset;
END_TRANSITION
STEP ModoReset:
    StopperOFF(N);
    FinPuesto(N);
END_STEP
TRANSITION FROM ModoReset TO EsperaPallet
    := not reset;
END_TRANSITION
STEP LiberaStoper:  // min time T#1s
    StopperOFF(N);
    ControlFallos(R);
END_STEP
TRANSITION FROM LiberaStoper TO Init
    := Not SensorPallet;
END_TRANSITION

ACTION ControlFallos:

IF GVL.FalloPallet[NumeroDePuesto] THEN
	LuzRoja :=TRUE;
	FinPuesto := FALSE;
ELSE
	LuzRoja :=FALSE;
	FinPuesto := TRUE;
END_IF


IF GVL.FalloPallet[NumeroDePuesto] AND Pulsador1 THEN
	GVL.FalloPallet[NumeroDePuesto] := FALSE;
END_IF
END_ACTION

ACTION Init_active:
LuzRoja := FALSE;
FinPUesto :=FALSE;
SFCreset:=FALSE;
END_ACTION

END_FUNCTION_BLOCK

// ---- POUs/PuestoCupula.TcPOU
FUNCTION_BLOCK PuestoCupula
VAR_INPUT
	Reset:BOOL;
	SFCreset:BOOL;
	Enable:BOOL;
	FinCiclo:BOOL;
	SensorPallet:BOOL;
	Pulsador1 AT %I*:BOOL;
	NumeroDePuesto :INT;	
	SelectorByPass AT %I*:BOOL;
	Pass AT %I*:BOOL;
	Fail AT %I*:BOOL;
	
	SensorPieza1 AT %I*:BOOL;
	SensorPieza2 AT %I*:BOOL;
	
	SensorCupulaAtras AT%I*:BOOL;

END_VAR
VAR_OUTPUT
	
	Ready AT %Q*:BOOL;
	StopperOFF AT %Q*:BOOL;
	Centrador AT%Q*:BOOL;
	Actuador AT%Q*:BOOL;
	LuzAmbar AT%Q*:BOOL;
	SalidaAlarma:BOOL;
	EnMovimiento:BOOL;
	EsperandoPalet:BOOL;
	RetrasoPuesto :INT;
	FinPuesto:BOOL;
	
	CupulaAdelante AT%Q*:BOOL;
	CupulaAtras AT%Q*:BOOL;

	
	
END_VAR

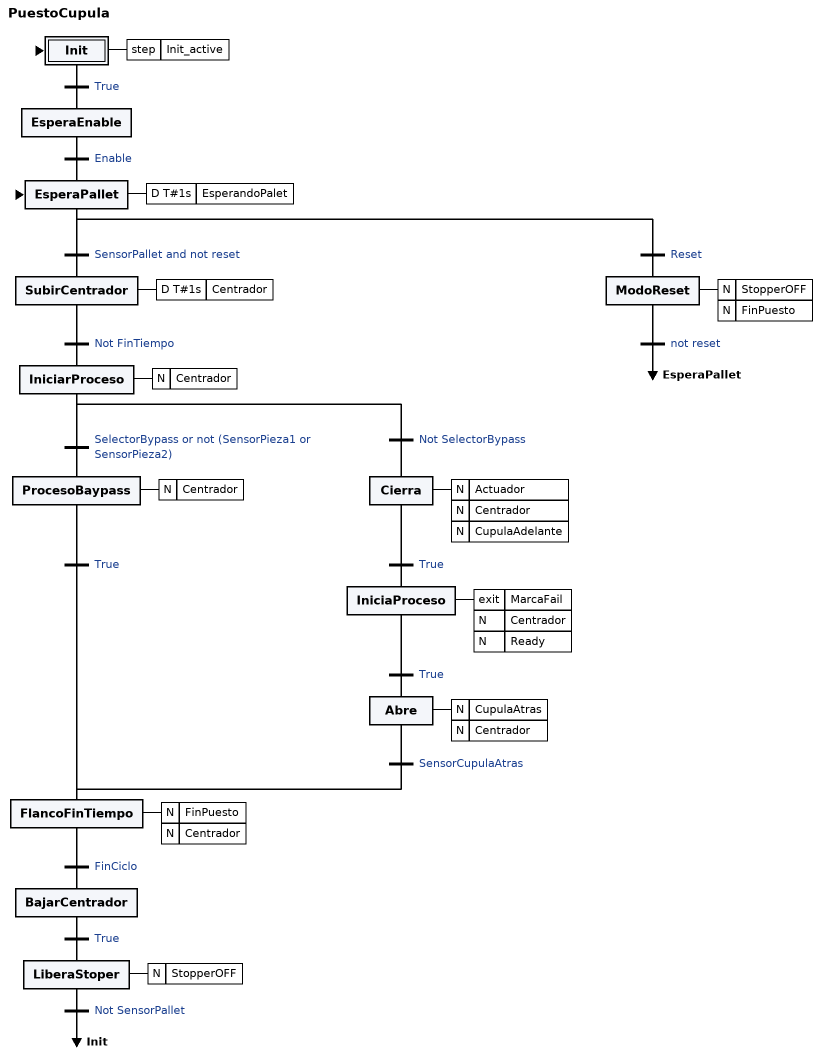
INITIAL_STEP Init:
    Init_active(N);  // step action
END_STEP
TRANSITION FROM Init TO EsperaEnable
    := True;
END_TRANSITION
STEP EsperaEnable:
END_STEP
TRANSITION FROM EsperaEnable TO EsperaPallet
    := Enable;
END_TRANSITION
STEP EsperaPallet:
    EsperandoPalet(D, T#1s);
END_STEP
TRANSITION FROM EsperaPallet TO SubirCentrador
    := SensorPallet and not reset;
END_TRANSITION
STEP SubirCentrador:  // min time T#2s
    Centrador(D, T#1s);
END_STEP
TRANSITION FROM SubirCentrador TO IniciarProceso
    := Not FinTiempo;
END_TRANSITION
STEP IniciarProceso:
    Centrador(N);
END_STEP
TRANSITION FROM IniciarProceso TO ProcesoBaypass
    := SelectorBypass or not (SensorPieza1 or SensorPieza2);
END_TRANSITION
STEP ProcesoBaypass:
    Centrador(N);
END_STEP
TRANSITION FROM ProcesoBaypass TO FlancoFinTiempo
    := True;
END_TRANSITION
TRANSITION FROM IniciarProceso TO Cierra
    := Not SelectorBypass;
END_TRANSITION
STEP Cierra:  // min time T#5s
    Actuador(N);
    Centrador(N);
    CupulaAdelante(N);
END_STEP
TRANSITION FROM Cierra TO IniciaProceso
    := True;
END_TRANSITION
STEP IniciaProceso:  // min time T#5s
    MarcaFail(P0);  // exit action
    Centrador(N);
    Ready(N);
END_STEP
TRANSITION FROM IniciaProceso TO Abre
    := True;
END_TRANSITION
STEP Abre:
    CupulaAtras(N);
    Centrador(N);
END_STEP
TRANSITION FROM Abre TO FlancoFinTiempo
    := SensorCupulaAtras;
END_TRANSITION
STEP FlancoFinTiempo:
    FinPuesto(N);
    Centrador(N);
END_STEP
TRANSITION FROM FlancoFinTiempo TO BajarCentrador
    := FinCiclo;
END_TRANSITION
STEP BajarCentrador:  // min time T#1s
END_STEP
TRANSITION FROM BajarCentrador TO LiberaStoper
    := True;
END_TRANSITION
TRANSITION FROM EsperaPallet TO ModoReset
    := Reset;
END_TRANSITION
STEP ModoReset:
    StopperOFF(N);
    FinPuesto(N);
END_STEP
TRANSITION FROM ModoReset TO EsperaPallet
    := not reset;
END_TRANSITION
STEP LiberaStoper:  // min time T#1s
    StopperOFF(N);
END_STEP
TRANSITION FROM LiberaStoper TO Init
    := Not SensorPallet;
END_TRANSITION

ACTION EsperaEnable_active:

END_ACTION

ACTION Init_active:
FinPUesto :=FALSE;
SFCreset:=FALSE;
END_ACTION

ACTION MarcaFail:
IF  Fail = TRUE THEN 
	gvl.FalloPallet[NumeroDePuesto] := TRUE;
END_IF
END_ACTION

END_FUNCTION_BLOCK

// ---- POUs/PuestoAutomatico.TcPOU
FUNCTION_BLOCK PuestoAutomatico
VAR_INPUT
	Reset:BOOL;
	SFCreset:BOOL;
	Enable:BOOL;
	FinCiclo:BOOL;
	SensorPallet:BOOL;
	Pulsador1 AT %I*:BOOL;

	NumeroDePuesto :INT;
	
	SelectorByPass AT %I*:BOOL;
	Pass AT %I*:BOOL;
	Fail AT %I*:BOOL;
	
	SensorPieza1 AT %I*:BOOL;
	SensorPieza2 AT %I*:BOOL;
	
END_VAR
VAR_OUTPUT
	
	Ready AT %Q*:BOOL;
	StopperOFF AT %Q*:BOOL;
	Centrador AT%Q*:BOOL;
	LuzAmbar AT%Q*:BOOL;
	SalidaAlarma:BOOL;
	EnMovimiento:BOOL;
	EsperandoPalet:BOOL;
	RetrasoPuesto :INT;
	FinPuesto:BOOL;
	
	
	
END_VAR
VAR
END_VAR

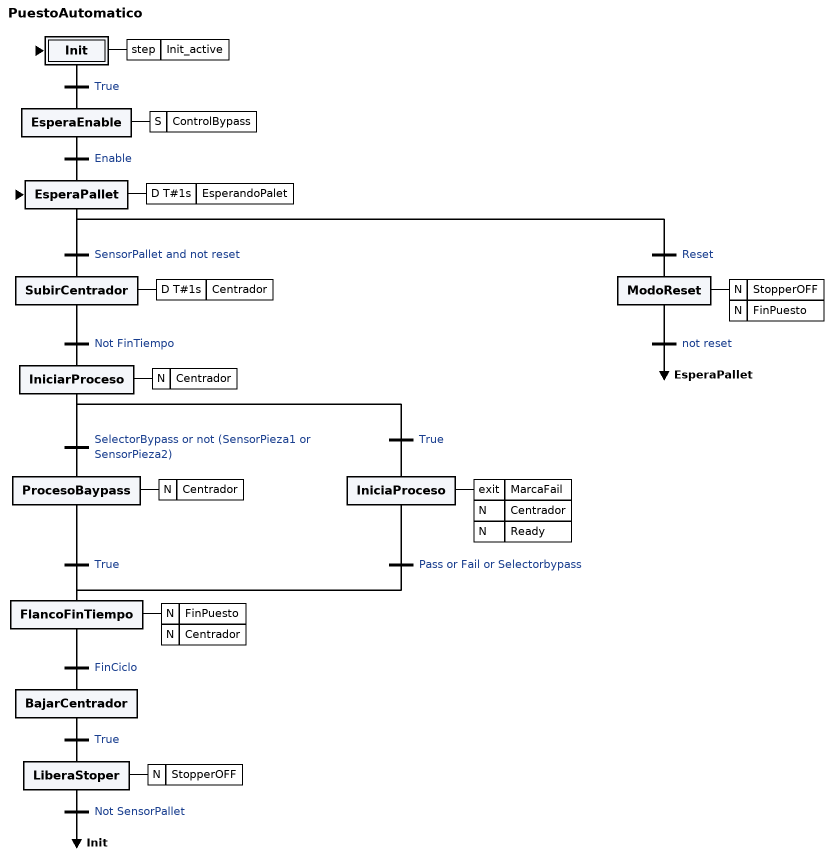
INITIAL_STEP Init:
    Init_active(N);  // step action
END_STEP
TRANSITION FROM Init TO EsperaEnable
    := True;
END_TRANSITION
STEP EsperaEnable:
    ControlBypass(S);
END_STEP
TRANSITION FROM EsperaEnable TO EsperaPallet
    := Enable;
END_TRANSITION
STEP EsperaPallet:
    EsperandoPalet(D, T#1s);
END_STEP
TRANSITION FROM EsperaPallet TO SubirCentrador
    := SensorPallet and not reset;
END_TRANSITION
STEP SubirCentrador:  // min time T#2s
    Centrador(D, T#1s);
END_STEP
TRANSITION FROM SubirCentrador TO IniciarProceso
    := Not FinTiempo;
END_TRANSITION
STEP IniciarProceso:
    Centrador(N);
END_STEP
TRANSITION FROM IniciarProceso TO ProcesoBaypass
    := SelectorBypass or not (SensorPieza1 or SensorPieza2);
END_TRANSITION
STEP ProcesoBaypass:
    Centrador(N);
END_STEP
TRANSITION FROM ProcesoBaypass TO FlancoFinTiempo
    := True;
END_TRANSITION
TRANSITION FROM IniciarProceso TO IniciaProceso
    := True;
END_TRANSITION
STEP IniciaProceso:
    MarcaFail(P0);  // exit action
    Centrador(N);
    Ready(N);
END_STEP
TRANSITION FROM IniciaProceso TO FlancoFinTiempo
    := Pass or Fail or Selectorbypass;
END_TRANSITION
STEP FlancoFinTiempo:
    FinPuesto(N);
    Centrador(N);
END_STEP
TRANSITION FROM FlancoFinTiempo TO BajarCentrador
    := FinCiclo;
END_TRANSITION
STEP BajarCentrador:  // min time T#1s
END_STEP
TRANSITION FROM BajarCentrador TO LiberaStoper
    := True;
END_TRANSITION
TRANSITION FROM EsperaPallet TO ModoReset
    := Reset;
END_TRANSITION
STEP ModoReset:
    StopperOFF(N);
    FinPuesto(N);
END_STEP
TRANSITION FROM ModoReset TO EsperaPallet
    := not reset;
END_TRANSITION
STEP LiberaStoper:  // min time T#1s
    StopperOFF(N);
END_STEP
TRANSITION FROM LiberaStoper TO Init
    := Not SensorPallet;
END_TRANSITION

ACTION ControlBypass:
LuzAmbar := SelectorByPass;
END_ACTION

ACTION Init_active:
FinPUesto :=FALSE;
SFCreset:=FALSE;
END_ACTION

ACTION MarcaFail:
IF  Fail = TRUE THEN 
	gvl.FalloPallet[NumeroDePuesto] := TRUE;
END_IF
END_ACTION

END_FUNCTION_BLOCK

// ---- POUs/PuestoManualV2.TcPOU
FUNCTION_BLOCK PuestoManualV2
VAR_INPUT
	SFCreset:BOOL;
	Reset:BOOL;
	Enable:BOOL;
	FinCiclo:BOOL;
	SensorPallet:BOOL;
	Pulsador1 AT %I*:BOOL;
	ModoDoble:BOOL;
	NumeroDePuesto :INT;
	
END_VAR
VAR_OUTPUT
	StopperOFF AT %Q*:BOOL;
	Centrador AT%Q*:BOOL;
	LuzRoja AT%Q*:BOOL;
	FinPuesto:BOOL;
	SalidaAlarma:BOOL;
	EnMovimiento:BOOL;
	EsperandoPalet :BOOL;
END_VAR
VAR
END_VAR

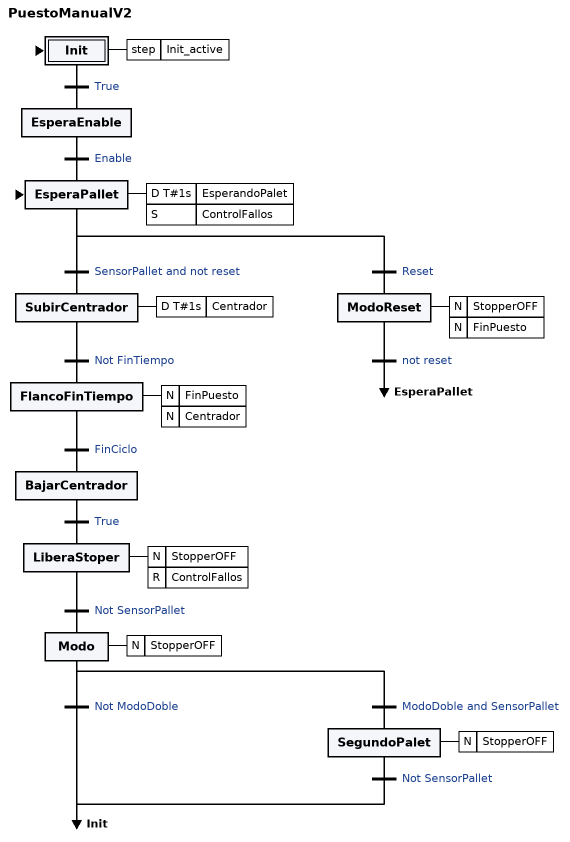
INITIAL_STEP Init:
    Init_active(N);  // step action
END_STEP
TRANSITION FROM Init TO EsperaEnable
    := True;
END_TRANSITION
STEP EsperaEnable:
END_STEP
TRANSITION FROM EsperaEnable TO EsperaPallet
    := Enable;
END_TRANSITION
STEP EsperaPallet:
    EsperandoPalet(D, T#1s);
    ControlFallos(S);
END_STEP
TRANSITION FROM EsperaPallet TO SubirCentrador
    := SensorPallet and not reset;
END_TRANSITION
STEP SubirCentrador:  // min time T#1s
    Centrador(D, T#1s);
END_STEP
TRANSITION FROM SubirCentrador TO FlancoFinTiempo
    := Not FinTiempo;
END_TRANSITION
STEP FlancoFinTiempo:
    FinPuesto(N);
    Centrador(N);
END_STEP
TRANSITION FROM FlancoFinTiempo TO BajarCentrador
    := FinCiclo;
END_TRANSITION
STEP BajarCentrador:  // min time T#1s
END_STEP
TRANSITION FROM BajarCentrador TO LiberaStoper
    := True;
END_TRANSITION
TRANSITION FROM EsperaPallet TO ModoReset
    := Reset;
END_TRANSITION
STEP ModoReset:
    StopperOFF(N);
    FinPuesto(N);
END_STEP
TRANSITION FROM ModoReset TO EsperaPallet
    := not reset;
END_TRANSITION
STEP LiberaStoper:  // min time T#1s
    StopperOFF(N);
    ControlFallos(R);
END_STEP
TRANSITION FROM LiberaStoper TO Modo
    := Not SensorPallet;
END_TRANSITION
STEP Modo:
    StopperOFF(N);
END_STEP
TRANSITION FROM Modo TO Init
    := Not ModoDoble;
END_TRANSITION
TRANSITION FROM Modo TO SegundoPalet
    := ModoDoble and SensorPallet;
END_TRANSITION
STEP SegundoPalet:  // min time T#1s
    StopperOFF(N);
END_STEP
TRANSITION FROM SegundoPalet TO Init
    := Not SensorPallet;
END_TRANSITION

ACTION ControlFallos:

IF GVL.FalloPallet[NumeroDePuesto] THEN
	LuzRoja :=TRUE;
	FinPuesto := FALSE;
ELSE
	LuzRoja :=TRUE;
	FinPuesto := FALSE;
END_IF


IF GVL.FalloPallet[NumeroDePuesto] AND Pulsador1 THEN
	GVL.FalloPallet[NumeroDePuesto] := FALSE;
END_IF
END_ACTION

ACTION Init_active:
LuzRoja := FALSE;
FinPUesto :=FALSE;
SFCreset:=FALSE;
END_ACTION

END_FUNCTION_BLOCK

// ---- POUs/ControlDescensoFin.TcPOU
FUNCTION_BLOCK ControlDescensoFin
VAR_INPUT
		SFCreset:BOOL;
	    SeguridadOK AT %I*: BOOL;
	    SensorArriba AT %I*: BOOL;
		SensorAbajo AT %I*:BOOL;
		Enabled AT %I*:BOOL;
		PuedeExtraer :BOOL;
		
		SensorPaletDentro AT %I*:BOOL;
		SensorPaletFuera AT %I*:BOOL;
		ElevadorLleno :BOOL;
		PulsadorBajar AT%I*: BOOL;
		PulsadorSubir AT%I*: BOOL;	

		PresenciaCintaArriba AT%I* :BOOL;
		PresenciaCintaAbajo AT %I* : BOOL;	
		
		ResetError :BOOL;
		
		MotorElevacion_Status AT%I*:UINT;
		MotorExtraccion_Status AT%I*:UINT;

END_VAR
VAR_OUTPUT
		MotorElevacion_Freq  AT%Q*: UINT;
	    MotorElevacion_Command AT%Q*: UINT;
		
		MotorExtraccion_Freq  AT%Q*: UINT;
	    MotorExtraccion_Command AT%Q*: UINT;
		
		Ready: BOOL; 
		
END_VAR
VAR
	VelocidadAlta :UINT := 4000;
	VelocidadBAJA :UINT := 1500;
	ModoVelocidadAlta :BOOL := FALSE;
	TiempoAltaVelocidad :TIME := T#3S;
	ERROR :BOOL;
	TimerEntradaSalida: TON;
	
	HomeOK :BOOL;
END_VAR

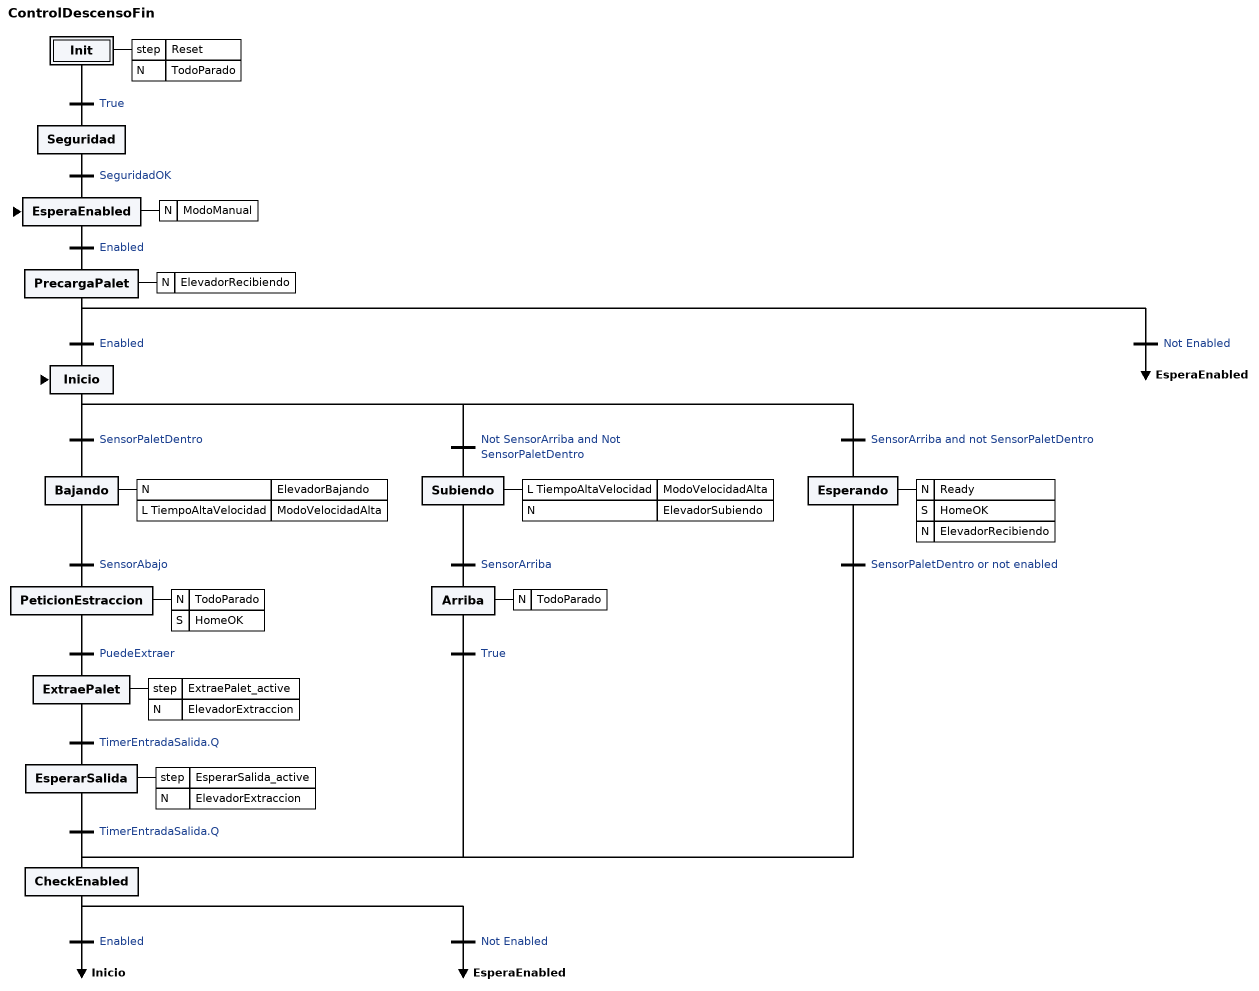
INITIAL_STEP Init:
    Reset(N);  // step action
    TodoParado(N);
END_STEP
TRANSITION FROM Init TO Seguridad
    := True;
END_TRANSITION
STEP Seguridad:
END_STEP
TRANSITION FROM Seguridad TO EsperaEnabled
    := SeguridadOK;
END_TRANSITION
STEP EsperaEnabled:
    ModoManual(N);
END_STEP
TRANSITION FROM EsperaEnabled TO PrecargaPalet
    := Enabled;
END_TRANSITION
STEP PrecargaPalet:  // min time T#2s
    ElevadorRecibiendo(N);
END_STEP
TRANSITION FROM PrecargaPalet TO Inicio
    := Enabled;
END_TRANSITION
TRANSITION FROM PrecargaPalet TO EsperaEnabled
    := Not Enabled;
END_TRANSITION
STEP Inicio:
END_STEP
TRANSITION FROM Inicio TO Bajando
    := SensorPaletDentro;
END_TRANSITION
STEP Bajando:
    ElevadorBajando(N);
    ModoVelocidadAlta(L, TiempoAltaVelocidad);
END_STEP
TRANSITION FROM Bajando TO PeticionEstraccion
    := SensorAbajo;
END_TRANSITION
STEP PeticionEstraccion:
    TodoParado(N);
    HomeOK(S);
END_STEP
TRANSITION FROM PeticionEstraccion TO ExtraePalet
    := PuedeExtraer;
END_TRANSITION
STEP ExtraePalet:  // min time T#1s
    ExtraePalet_active(N);  // step action
    ElevadorExtraccion(N);
END_STEP
TRANSITION FROM ExtraePalet TO EsperarSalida
    := TimerEntradaSalida.Q;
END_TRANSITION
STEP EsperarSalida:
    EsperarSalida_active(N);  // step action
    ElevadorExtraccion(N);
END_STEP
TRANSITION FROM EsperarSalida TO CheckEnabled
    := TimerEntradaSalida.Q;
END_TRANSITION
TRANSITION FROM Inicio TO Subiendo
    := Not SensorArriba and Not SensorPaletDentro;
END_TRANSITION
STEP Subiendo:
    ModoVelocidadAlta(L, TiempoAltaVelocidad);
    ElevadorSubiendo(N);
END_STEP
TRANSITION FROM Subiendo TO Arriba
    := SensorArriba;
END_TRANSITION
STEP Arriba:
    TodoParado(N);
END_STEP
TRANSITION FROM Arriba TO CheckEnabled
    := True;
END_TRANSITION
TRANSITION FROM Inicio TO Esperando
    := SensorArriba and not SensorPaletDentro;
END_TRANSITION
STEP Esperando:
    Ready(N);
    HomeOK(S);
    ElevadorRecibiendo(N);
END_STEP
TRANSITION FROM Esperando TO CheckEnabled
    := SensorPaletDentro or not enabled;
END_TRANSITION
STEP CheckEnabled:
END_STEP
TRANSITION FROM CheckEnabled TO Inicio
    := Enabled;
END_TRANSITION
TRANSITION FROM CheckEnabled TO EsperaEnabled
    := Not Enabled;
END_TRANSITION

ACTION ElevadorBajando:
MotorElevador(2);
MotorExtraccion(0);
END_ACTION

ACTION ElevadorExtraccion:

IF PuedeExtraer THEN
	MotorExtraccion(1);
ELSE 
	MotorExtraccion(0);
END_IF
END_ACTION

ACTION ElevadorRecibiendo:
MotorElevador(0);

IF Enabled THEN
	MotorExtraccion(2);
ELSE 
	MotorExtraccion(0);
END_IF
END_ACTION

ACTION ElevadorSubiendo:
MotorElevador(1);
MotorExtraccion(0);
END_ACTION

ACTION EsperarSalida_active:
TimerEntradaSalida(IN:=NOT PresenciaCintaAbajo, PT:= T#1S);
END_ACTION

ACTION ExtraePalet_active:
TimerEntradaSalida(IN:=PresenciaCintaAbajo, PT:= T#1S);
END_ACTION

ACTION ModoManual:


IF PulsadorSubir THEN
	MotorElevador(1);
		HomeOK :=FALSE;
ELSIF PulsadorBajar THEN
	MotorElevador(2);
		HomeOK :=FALSE;
ELSE
	MotorElevador(0);
END_IF
END_ACTION

METHOD PRIVATE MotorElevador : BOOL
VAR_INPUT
	Direccion : INT; //0 parado 1 subir 2 bajar
END_VAR
IF ModoVelocidadAlta AND HomeOK THEN
	MotorElevacion_Freq := 5000;
ELSE
	MotorElevacion_Freq := 1000;
END_IF


MotorElevacion_Command := 0;
MotorElevacion_Command.7 := 1 ; //Control Word Active

IF Direccion = 0 THEN
	MotorElevacion_Command.3 := 1 ; // Stop according to parameter setting	
ELSIF PresenciaCintaArriba OR PresenciaCintaAbajo THEN
	//ERROR: intenta mover elevador con obstatuclos
	//DEBE MOStrar error
	MotorElevacion_Command.3 := 1 ; // Stop according to parameter setting	
	
ELSIF Direccion  = 1 THEN
		
		MotorElevacion_Command.2 := 0 ; //1 reversed 0 fordward
		MotorElevacion_Command.0 := 1 ; // Run Command active
		HomeOK :=FALSE;

ELSIF Direccion= 2 THEN
	MotorElevacion_Command.2 := 1 ; //1 reversed 0 fordward
	MotorElevacion_Command.0 := 1 ; // Run Command active
		HomeOK :=FALSE;
ELSE
	MotorElevacion_Command.3 := 1 ; // Stop according to parameter setting	
END_IF
END_METHOD

METHOD PRIVATE MotorExtraccion : BOOL
VAR_INPUT
	Direccion : INT; //0 parado 1 salida 2 entrada
END_VAR

MotorExtraccion_Freq := gvl.VelocidadCinta * 100;
MotorExtraccion_Command := 0;
MotorExtraccion_Command.7 := 1 ; //Control Word Active

IF Direccion  = 1 THEN
	MotorExtraccion_Command.2 := 1 ; //1 reversed 0 fordward
	MotorExtraccion_Command.0 := 1 ; // Run Command active
ELSIF Direccion= 2 THEN
	MotorExtraccion_Command.2 := 0 ; //1 reversed 0 fordward
	MotorExtraccion_Command.0 := 1 ; // Run Command active
ELSE
	MotorExtraccion_Command.3 := 1 ; // Stop according to parameter setting	
END_IF
END_METHOD

ACTION RealizaHome:
MotorElevador(1);
MotorExtraccion(0);
END_ACTION

ACTION Reset:
HomeOK := FALSE;
SFCreset:=FALSE;
END_ACTION

ACTION TodoParado:
MotorElevador(0);
MotorExtraccion(0);
END_ACTION

END_FUNCTION_BLOCK

// ---- POUs/ControlElevadorInicio.TcPOU
FUNCTION_BLOCK ControlElevadorInicio
VAR_INPUT
		SFCreset:BOOL;
	    SeguridadOK : BOOL;
	    SensorArriba AT %I*: BOOL;
		SensorAbajo AT %I*:BOOL;
		Enabled AT %I*:BOOL;
		
		SensorPaletDentro AT %I*:BOOL;
		SensorPaletFuera AT %I*:BOOL;
		SensorPaletEnEspera AT %I*:BOOL;


		PulsadorBajar AT%I*: BOOL;
		PulsadorSubir AT%I*: BOOL;
		
		ResetError :BOOL;
		
		MotorElevacion_Status AT%I*:UINT;
		MotorExtraccion_Status AT%I*:UINT;

		PuedeExtraer :BOOL;
END_VAR
VAR_OUTPUT
		MotorElevacion_Freq  AT%Q*: UINT;
	    MotorElevacion_Command AT%Q*: INT;
		
		MotorExtraccion_Freq  AT%Q*: UINT;
	    MotorExtraccion_Command AT%Q*: INT;
		
		StopperOFF AT %Q*: BOOL;
		
		PresenciaCintaArriba AT%I* :BOOL;
		PresenciaCintaAbajo AT %I* : BOOL;	
		
		Ready: BOOL;
		EsperandoPalet :BOOL;
		
END_VAR
VAR
	VelocidadAlta :UINT := 4000;
	VelocidadBAJA :UINT := 1500;
	ModoVelocidadAlta :BOOL := FALSE;
	TiempoAltaVelocidad :TIME := T#3S;
	
	ERROR :BOOL;
	PosicionArriba: WORD := 141;

	HomeOk :BOOL;
END_VAR

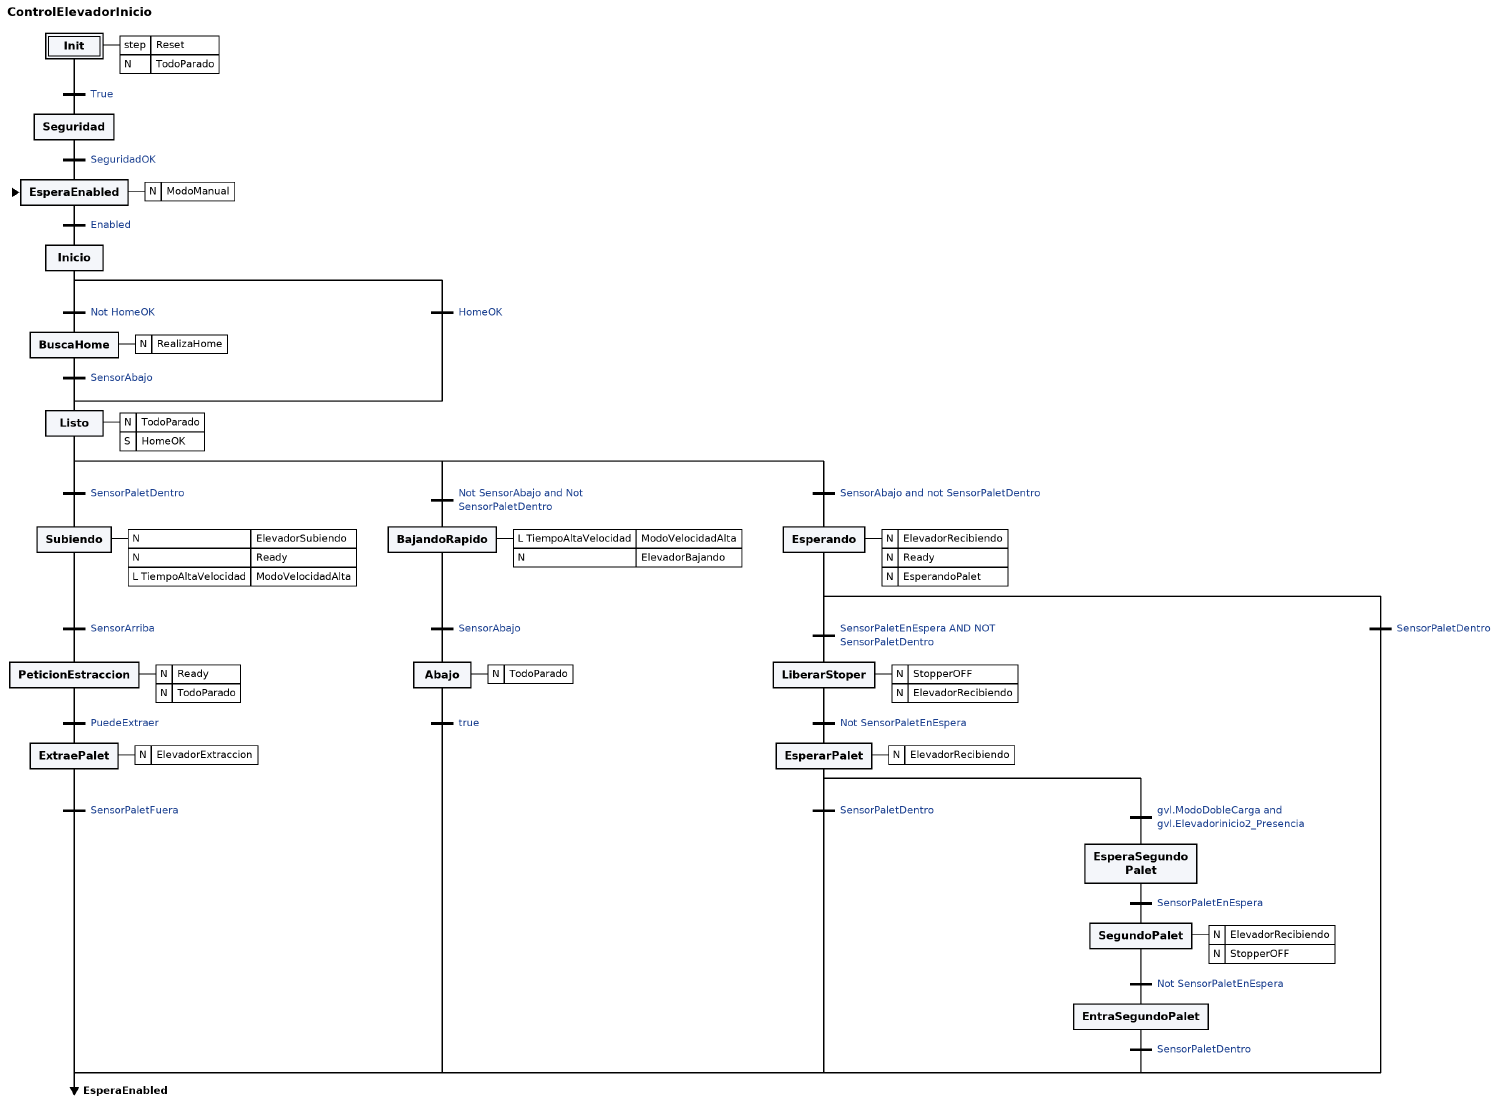
INITIAL_STEP Init:
    Reset(N);  // step action
    TodoParado(N);
END_STEP
TRANSITION FROM Init TO Seguridad
    := True;
END_TRANSITION
STEP Seguridad:
END_STEP
TRANSITION FROM Seguridad TO EsperaEnabled
    := SeguridadOK;
END_TRANSITION
STEP EsperaEnabled:
    ModoManual(N);
END_STEP
TRANSITION FROM EsperaEnabled TO Inicio
    := Enabled;
END_TRANSITION
STEP Inicio:
END_STEP
TRANSITION FROM Inicio TO BuscaHome
    := Not HomeOK;
END_TRANSITION
STEP BuscaHome:
    RealizaHome(N);
END_STEP
TRANSITION FROM BuscaHome TO Listo
    := SensorAbajo;
END_TRANSITION
TRANSITION FROM Inicio TO Listo
    := HomeOK;
END_TRANSITION
STEP Listo:
    TodoParado(N);
    HomeOK(S);
END_STEP
TRANSITION FROM Listo TO Subiendo
    := SensorPaletDentro;
END_TRANSITION
STEP Subiendo:
    ElevadorSubiendo(N);
    Ready(N);
    ModoVelocidadAlta(L, TiempoAltaVelocidad);
END_STEP
TRANSITION FROM Subiendo TO PeticionEstraccion
    := SensorArriba;
END_TRANSITION
STEP PeticionEstraccion:
    Ready(N);
    TodoParado(N);
END_STEP
TRANSITION FROM PeticionEstraccion TO ExtraePalet
    := PuedeExtraer;
END_TRANSITION
STEP ExtraePalet:
    ElevadorExtraccion(N);
END_STEP
TRANSITION FROM ExtraePalet TO EsperaEnabled
    := SensorPaletFuera;
END_TRANSITION
TRANSITION FROM Listo TO BajandoRapido
    := Not SensorAbajo and Not SensorPaletDentro;
END_TRANSITION
STEP BajandoRapido:
    ModoVelocidadAlta(L, TiempoAltaVelocidad);
    ElevadorBajando(N);
END_STEP
TRANSITION FROM BajandoRapido TO Abajo
    := SensorAbajo;
END_TRANSITION
STEP Abajo:
    TodoParado(N);
END_STEP
TRANSITION FROM Abajo TO EsperaEnabled
    := true;
END_TRANSITION
TRANSITION FROM Listo TO Esperando
    := SensorAbajo and not SensorPaletDentro;
END_TRANSITION
STEP Esperando:  // min time T#1s
    ElevadorRecibiendo(N);
    Ready(N);
    EsperandoPalet(N);
END_STEP
TRANSITION FROM Esperando TO LiberarStoper
    := SensorPaletEnEspera AND NOT SensorPaletDentro;
END_TRANSITION
STEP LiberarStoper:
    StopperOFF(N);
    ElevadorRecibiendo(N);
END_STEP
TRANSITION FROM LiberarStoper TO EsperarPalet
    := Not SensorPaletEnEspera;
END_TRANSITION
STEP EsperarPalet:
    ElevadorRecibiendo(N);
END_STEP
TRANSITION FROM EsperarPalet TO EsperaEnabled
    := SensorPaletDentro;
END_TRANSITION
TRANSITION FROM EsperarPalet TO EsperaSegundoPalet
    := gvl.ModoDobleCarga and gvl.Elevadorinicio2_Presencia;
END_TRANSITION
STEP EsperaSegundoPalet:
END_STEP
TRANSITION FROM EsperaSegundoPalet TO SegundoPalet
    := SensorPaletEnEspera;
END_TRANSITION
STEP SegundoPalet:
    ElevadorRecibiendo(N);
    StopperOFF(N);
END_STEP
TRANSITION FROM SegundoPalet TO EntraSegundoPalet
    := Not SensorPaletEnEspera;
END_TRANSITION
STEP EntraSegundoPalet:
END_STEP
TRANSITION FROM EntraSegundoPalet TO EsperaEnabled
    := SensorPaletDentro;
END_TRANSITION
TRANSITION FROM Esperando TO EsperaEnabled
    := SensorPaletDentro;
END_TRANSITION

ACTION ElevadorBajando:
MotorElevador(2);
MotorExtraccion(0);
END_ACTION

ACTION ElevadorExtraccion:

IF PuedeExtraer THEN
	MotorExtraccion(1);
ELSE 
	MotorExtraccion(0);
END_IF
END_ACTION

ACTION ElevadorRecibiendo:
MotorElevador(0);

IF Enabled THEN
	MotorExtraccion(2);
ELSE 
	MotorExtraccion(0);
END_IF
END_ACTION

ACTION ElevadorSubiendo:
MotorElevador(1);
MotorExtraccion(0);
END_ACTION

ACTION ModoManual:

IF PulsadorSubir THEN
		MotorElevador(1);
		HomeOK :=FALSE;
ELSIF PulsadorBajar THEN
		MotorElevador(2);
		HomeOK :=FALSE;
ELSE
		MotorElevador(0);	
END_IF
END_ACTION

METHOD PRIVATE MotorElevador : BOOL
VAR_INPUT
	Direccion : INT; //0 parado 1 subir 2 bajar
END_VAR
IF ModoVelocidadAlta THEN
	MotorElevacion_Freq := 5000;
ELSE
	MotorElevacion_Freq := 1000;
END_IF


MotorElevacion_Command := 0;
MotorElevacion_Command.7 := 1 ; //Control Word Active

IF Direccion = 0 THEN
	MotorElevacion_Command.3 := 1 ; // Stop according to parameter setting	
ELSIF PresenciaCintaArriba OR PresenciaCintaAbajo THEN
	//ERROR: intenta mover elevador con obstatuclos
	//DEBE MOStrar error
	MotorElevacion_Command.3 := 1 ; // Stop according to parameter setting	
ELSIF Direccion  = 1 THEN
	MotorElevacion_Command.2 := 0 ; //1 reversed 0 fordward
	MotorElevacion_Command.0 := 1 ; // Run Command active
		HomeOK :=FALSE;
ELSIF Direccion= 2 THEN
	MotorElevacion_Command.2 := 1 ; //1 reversed 0 fordward
	MotorElevacion_Command.0 := 1 ; // Run Command active
		HomeOK :=FALSE;
ELSE
	MotorElevacion_Command.3 := 1 ; // Stop according to parameter setting	
END_IF
END_METHOD

METHOD PRIVATE MotorExtraccion : BOOL
VAR_INPUT
	Direccion : INT; //0 parado 1 salida 2 entrada
END_VAR

MotorExtraccion_Freq := gvl.VelocidadCinta * 100;
MotorExtraccion_Command := 0;
MotorExtraccion_Command.7 := 1 ; //Control Word Active

IF Direccion  = 1 THEN
	MotorExtraccion_Command.2 := 0 ; //1 reversed 0 fordward
	MotorExtraccion_Command.0 := 1 ; // Run Command active
ELSIF Direccion= 2 THEN
	MotorExtraccion_Command.2 := 1 ; //1 reversed 0 fordward
	MotorExtraccion_Command.0 := 1 ; // Run Command active
ELSE
	MotorExtraccion_Command.3 := 1 ; // Stop according to parameter setting	
END_IF
END_METHOD

ACTION RealizaHome:
MotorElevador(2);
MotorExtraccion(0);
END_ACTION

ACTION Reset:
HomeOK := FALSE;
SFCreset:=FALSE;
END_ACTION

ACTION TodoParado:
MotorElevador(0);
MotorExtraccion(0);
END_ACTION

END_FUNCTION_BLOCK

// ---- POUs/PuestoTester.TcPOU
FUNCTION_BLOCK PuestoTester
VAR_INPUT
	Reset:BOOL;
	SFCreset:BOOL;
	Enable:BOOL;
	FinCiclo:BOOL;
	SensorPallet:BOOL;
	Pulsador1 AT %I*:BOOL;
	NumeroDePuesto :INT;	
	SelectorByPass AT %I*:BOOL;
	Pass AT %I*:BOOL;
	Fail AT %I*:BOOL;
	
	SensorPieza1 AT %I*:BOOL;
	SensorPieza2 AT %I*:BOOL;
	
END_VAR
VAR_OUTPUT
	
	Ready AT %Q*:BOOL;
	StopperOFF AT %Q*:BOOL;
	Centrador AT%Q*:BOOL;
	Actuador AT%Q*:BOOL;
	LuzAmbar AT%Q*:BOOL;
	SalidaAlarma:BOOL;
	EnMovimiento:BOOL;
	EsperandoPalet:BOOL;
	RetrasoPuesto :INT;
	FinPuesto:BOOL;
	
	
	
END_VAR

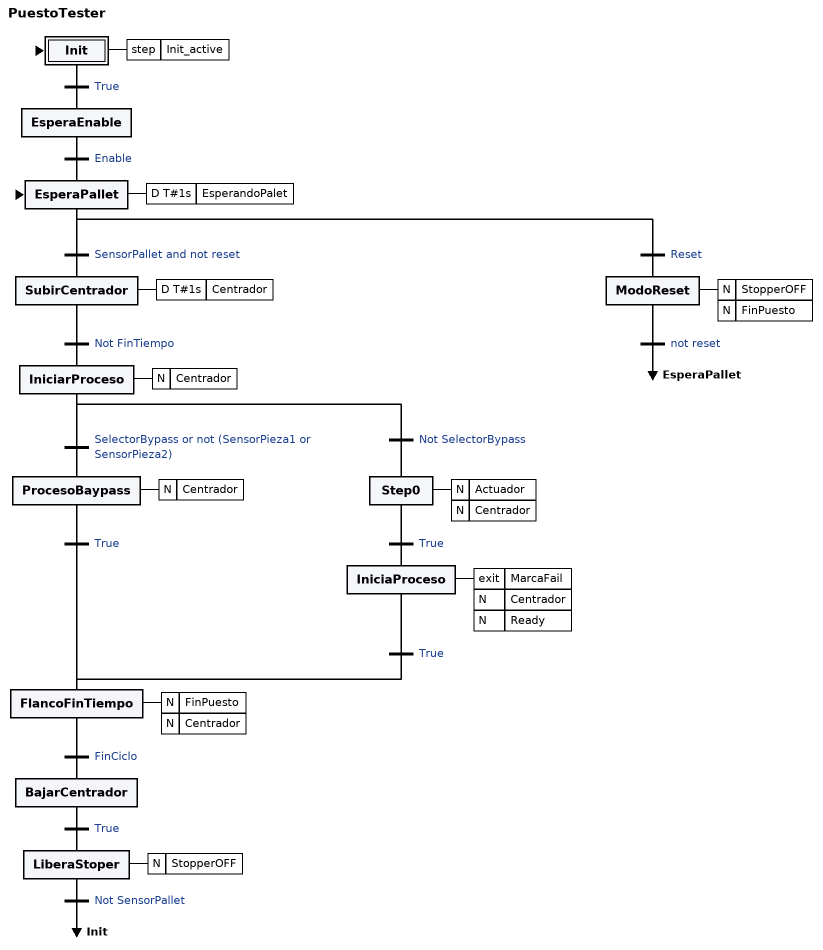
INITIAL_STEP Init:
    Init_active(N);  // step action
END_STEP
TRANSITION FROM Init TO EsperaEnable
    := True;
END_TRANSITION
STEP EsperaEnable:
END_STEP
TRANSITION FROM EsperaEnable TO EsperaPallet
    := Enable;
END_TRANSITION
STEP EsperaPallet:
    EsperandoPalet(D, T#1s);
END_STEP
TRANSITION FROM EsperaPallet TO SubirCentrador
    := SensorPallet and not reset;
END_TRANSITION
STEP SubirCentrador:  // min time T#2s
    Centrador(D, T#1s);
END_STEP
TRANSITION FROM SubirCentrador TO IniciarProceso
    := Not FinTiempo;
END_TRANSITION
STEP IniciarProceso:
    Centrador(N);
END_STEP
TRANSITION FROM IniciarProceso TO ProcesoBaypass
    := SelectorBypass or not (SensorPieza1 or SensorPieza2);
END_TRANSITION
STEP ProcesoBaypass:
    Centrador(N);
END_STEP
TRANSITION FROM ProcesoBaypass TO FlancoFinTiempo
    := True;
END_TRANSITION
TRANSITION FROM IniciarProceso TO Step0
    := Not SelectorBypass;
END_TRANSITION
STEP Step0:  // min time T#5s
    Actuador(N);
    Centrador(N);
END_STEP
TRANSITION FROM Step0 TO IniciaProceso
    := True;
END_TRANSITION
STEP IniciaProceso:  // min time T#1s
    MarcaFail(P0);  // exit action
    Centrador(N);
    Ready(N);
END_STEP
TRANSITION FROM IniciaProceso TO FlancoFinTiempo
    := True;
END_TRANSITION
STEP FlancoFinTiempo:
    FinPuesto(N);
    Centrador(N);
END_STEP
TRANSITION FROM FlancoFinTiempo TO BajarCentrador
    := FinCiclo;
END_TRANSITION
STEP BajarCentrador:  // min time T#1s
END_STEP
TRANSITION FROM BajarCentrador TO LiberaStoper
    := True;
END_TRANSITION
TRANSITION FROM EsperaPallet TO ModoReset
    := Reset;
END_TRANSITION
STEP ModoReset:
    StopperOFF(N);
    FinPuesto(N);
END_STEP
TRANSITION FROM ModoReset TO EsperaPallet
    := not reset;
END_TRANSITION
STEP LiberaStoper:  // min time T#1s
    StopperOFF(N);
END_STEP
TRANSITION FROM LiberaStoper TO Init
    := Not SensorPallet;
END_TRANSITION

ACTION EsperaEnable_active:

END_ACTION

ACTION Init_active:
FinPUesto :=FALSE;
SFCreset:=FALSE;
END_ACTION

ACTION MarcaFail:
IF  Fail = TRUE THEN 
	gvl.FalloPallet[NumeroDePuesto] := TRUE;
END_IF
END_ACTION

END_FUNCTION_BLOCK
